// TIA Portal V19 export
FUNCTION "CEB_2" : Void   // FC15, LAD
{ S7_Optimized_Access := 'TRUE' }
// stored: SetENOAutomatically false
BEGIN

REGION Network 2: CEB_2 START
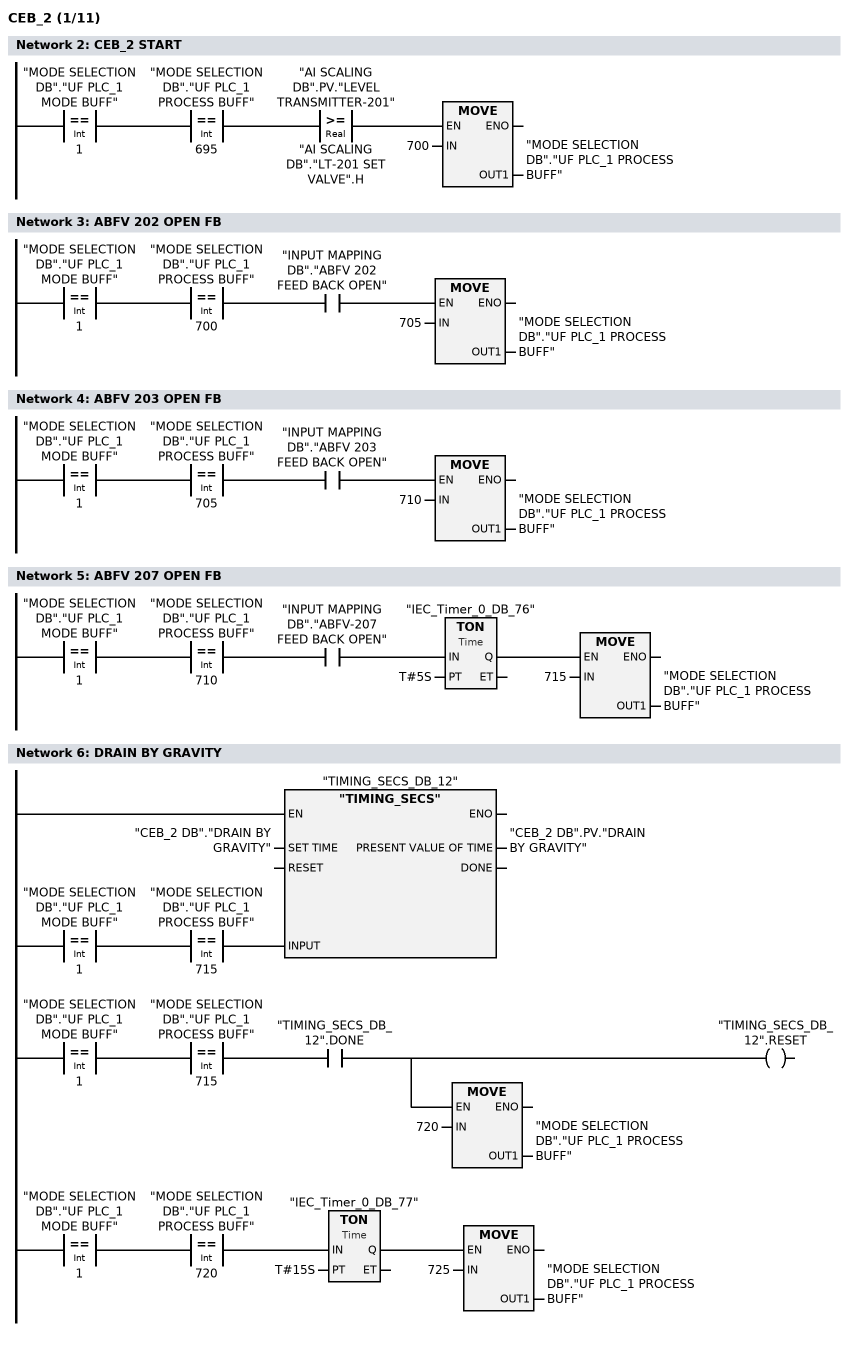
   RUNG wire#powerrail
      { S7_Templates := "SrcType := Int" } EQ_Contact(in1 := "MODE SELECTION DB"."UF PLC_1 MODE BUFF", in2 := 1)
      { S7_Templates := "SrcType := Int" } EQ_Contact(in1 := "MODE SELECTION DB"."UF PLC_1 PROCESS BUFF", in2 := 695)
      { S7_Templates := "SrcType := Real" } GE_Contact(in1 := "AI SCALING DB".PV."LEVEL TRANSMITTER-201", in2 := "AI SCALING DB"."LT-201 SET VALVE".H)
      Move(in := 700, out1 => "MODE SELECTION DB"."UF PLC_1 PROCESS BUFF")
   END_RUNG
   // the same network as SCL:
   IF ("MODE SELECTION DB"."UF PLC_1 MODE BUFF" = 1) AND ("MODE SELECTION DB"."UF PLC_1 PROCESS BUFF" = 695) AND ("AI SCALING DB".PV."LEVEL TRANSMITTER-201" >= "AI SCALING DB"."LT-201 SET VALVE".H) THEN
       "MODE SELECTION DB"."UF PLC_1 PROCESS BUFF" := 700;
   END_IF;
END_REGION

REGION Network 3: ABFV 202 OPEN FB
   RUNG wire#powerrail
      { S7_Templates := "SrcType := Int" } EQ_Contact(in1 := "MODE SELECTION DB"."UF PLC_1 MODE BUFF", in2 := 1)
      { S7_Templates := "SrcType := Int" } EQ_Contact(in1 := "MODE SELECTION DB"."UF PLC_1 PROCESS BUFF", in2 := 700)
      Contact( "INPUT MAPPING DB"."ABFV 202 FEED BACK OPEN" )
      Move(in := 705, out1 => "MODE SELECTION DB"."UF PLC_1 PROCESS BUFF")
   END_RUNG
   // the same network as SCL:
   IF ("MODE SELECTION DB"."UF PLC_1 MODE BUFF" = 1) AND ("MODE SELECTION DB"."UF PLC_1 PROCESS BUFF" = 700) AND "INPUT MAPPING DB"."ABFV 202 FEED BACK OPEN" THEN
       "MODE SELECTION DB"."UF PLC_1 PROCESS BUFF" := 705;
   END_IF;
END_REGION

REGION Network 4: ABFV 203 OPEN FB
   RUNG wire#powerrail
      { S7_Templates := "SrcType := Int" } EQ_Contact(in1 := "MODE SELECTION DB"."UF PLC_1 MODE BUFF", in2 := 1)
      { S7_Templates := "SrcType := Int" } EQ_Contact(in1 := "MODE SELECTION DB"."UF PLC_1 PROCESS BUFF", in2 := 705)
      Contact( "INPUT MAPPING DB"."ABFV 203 FEED BACK OPEN" )
      Move(in := 710, out1 => "MODE SELECTION DB"."UF PLC_1 PROCESS BUFF")
   END_RUNG
   // the same network as SCL:
   IF ("MODE SELECTION DB"."UF PLC_1 MODE BUFF" = 1) AND ("MODE SELECTION DB"."UF PLC_1 PROCESS BUFF" = 705) AND "INPUT MAPPING DB"."ABFV 203 FEED BACK OPEN" THEN
       "MODE SELECTION DB"."UF PLC_1 PROCESS BUFF" := 710;
   END_IF;
END_REGION

REGION Network 5: ABFV 207 OPEN FB
   RUNG wire#powerrail
      { S7_Templates := "SrcType := Int" } EQ_Contact(in1 := "MODE SELECTION DB"."UF PLC_1 MODE BUFF", in2 := 1)
      { S7_Templates := "SrcType := Int" } EQ_Contact(in1 := "MODE SELECTION DB"."UF PLC_1 PROCESS BUFF", in2 := 710)
      Contact( "INPUT MAPPING DB"."ABFV-207 FEED BACK OPEN" )
      { S7_Templates := "time_type := Time" } "IEC_Timer_0_DB_76".TON(pt := T#5S, et =>)
      Move(in := 715, out1 => "MODE SELECTION DB"."UF PLC_1 PROCESS BUFF")
   END_RUNG
   // the same network as SCL:
   "IEC_Timer_0_DB_76".TON(IN := ("MODE SELECTION DB"."UF PLC_1 MODE BUFF" = 1) AND ("MODE SELECTION DB"."UF PLC_1 PROCESS BUFF" = 710) AND "INPUT MAPPING DB"."ABFV-207 FEED BACK OPEN",
                           PT := T#5S);
   IF "IEC_Timer_0_DB_76".Q THEN "MODE SELECTION DB"."UF PLC_1 PROCESS BUFF" := 715; END_IF;
END_REGION

REGION Network 6: DRAIN BY GRAVITY
   RUNG wire#powerrail
      "TIMING_SECS_DB_12"(INPUT := wire#w1, "SET TIME" := "CEB_2 DB"."DRAIN BY GRAVITY", RESET :=, "PRESENT VALUE OF TIME" => "CEB_2 DB".PV."DRAIN BY GRAVITY", DONE =>)
   END_RUNG
   RUNG wire#powerrail
      { S7_Templates := "SrcType := Int" } EQ_Contact(in1 := "MODE SELECTION DB"."UF PLC_1 MODE BUFF", in2 := 1)
      { S7_Templates := "SrcType := Int" } EQ_Contact(in1 := "MODE SELECTION DB"."UF PLC_1 PROCESS BUFF", in2 := 715)
   END_RUNG wire#w1
   RUNG wire#powerrail
      { S7_Templates := "SrcType := Int" } EQ_Contact(in1 := "MODE SELECTION DB"."UF PLC_1 MODE BUFF", in2 := 1)
      { S7_Templates := "SrcType := Int" } EQ_Contact(in1 := "MODE SELECTION DB"."UF PLC_1 PROCESS BUFF", in2 := 715)
      Contact( "TIMING_SECS_DB_12".DONE )
      wire#w2
      Coil( "TIMING_SECS_DB_12".RESET )
   END_RUNG
   RUNG wire#w2
      Move(in := 720, out1 => "MODE SELECTION DB"."UF PLC_1 PROCESS BUFF")
   END_RUNG
   RUNG wire#powerrail
      { S7_Templates := "SrcType := Int" } EQ_Contact(in1 := "MODE SELECTION DB"."UF PLC_1 MODE BUFF", in2 := 1)
      { S7_Templates := "SrcType := Int" } EQ_Contact(in1 := "MODE SELECTION DB"."UF PLC_1 PROCESS BUFF", in2 := 720)
      { S7_Templates := "time_type := Time" } "IEC_Timer_0_DB_77".TON(pt := T#15S, et =>)
      Move(in := 725, out1 => "MODE SELECTION DB"."UF PLC_1 PROCESS BUFF")
   END_RUNG
   // the same network as SCL:
   "TIMING_SECS_DB_12"("SET TIME" := "CEB_2 DB"."DRAIN BY GRAVITY",   // "TIMING_SECS"
                       INPUT := ("MODE SELECTION DB"."UF PLC_1 MODE BUFF" = 1) AND ("MODE SELECTION DB"."UF PLC_1 PROCESS BUFF" = 715),
                       "PRESENT VALUE OF TIME" => "CEB_2 DB".PV."DRAIN BY GRAVITY");
   "TIMING_SECS_DB_12".RESET := ("MODE SELECTION DB"."UF PLC_1 MODE BUFF" = 1) AND ("MODE SELECTION DB"."UF PLC_1 PROCESS BUFF" = 715) AND "TIMING_SECS_DB_12".DONE;
   IF "TIMING_SECS_DB_12".RESET THEN "MODE SELECTION DB"."UF PLC_1 PROCESS BUFF" := 720; END_IF;
   "IEC_Timer_0_DB_77".TON(IN := ("MODE SELECTION DB"."UF PLC_1 MODE BUFF" = 1) AND ("MODE SELECTION DB"."UF PLC_1 PROCESS BUFF" = 720),
                           PT := T#15S);
   IF "IEC_Timer_0_DB_77".Q THEN "MODE SELECTION DB"."UF PLC_1 PROCESS BUFF" := 725; END_IF;
END_REGION

REGION Network 7: ABFV 207 CLOSE FB
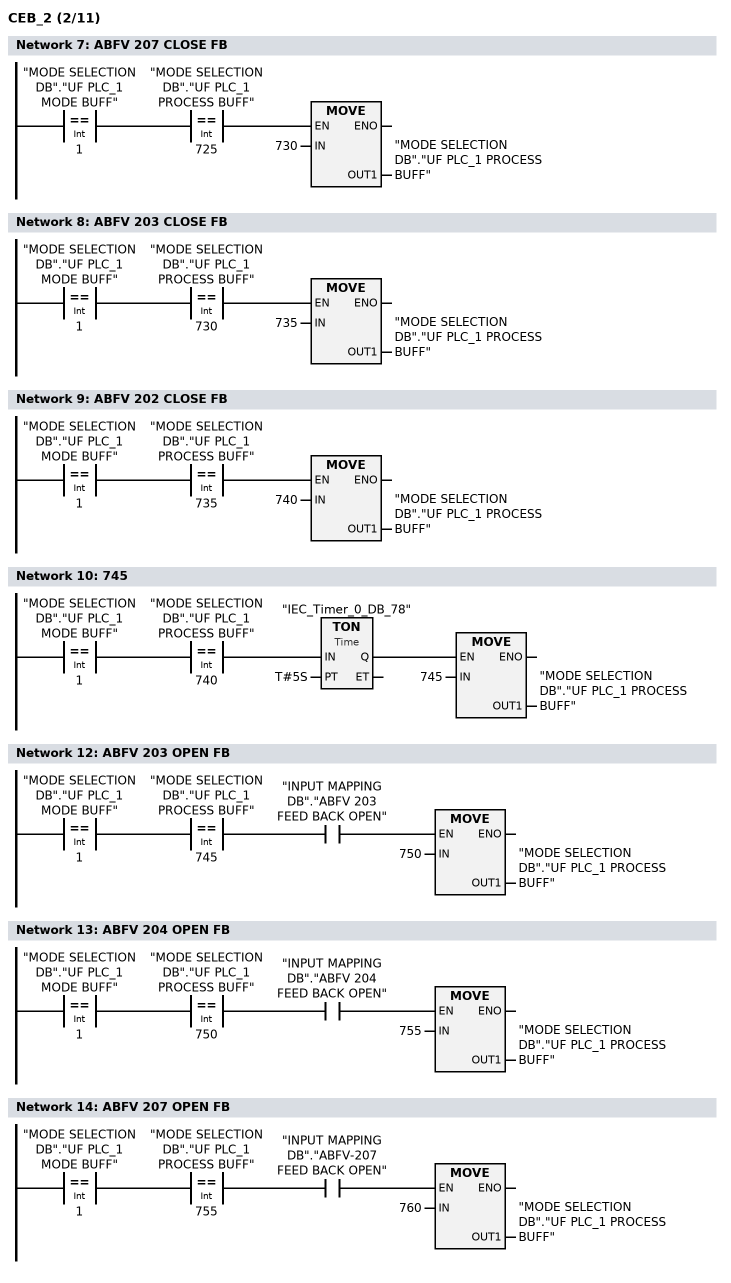
   RUNG wire#powerrail
      { S7_Templates := "SrcType := Int" } EQ_Contact(in1 := "MODE SELECTION DB"."UF PLC_1 MODE BUFF", in2 := 1)
      { S7_Templates := "SrcType := Int" } EQ_Contact(in1 := "MODE SELECTION DB"."UF PLC_1 PROCESS BUFF", in2 := 725)
      Move(in := 730, out1 => "MODE SELECTION DB"."UF PLC_1 PROCESS BUFF")
   END_RUNG
   // the same network as SCL:
   IF ("MODE SELECTION DB"."UF PLC_1 MODE BUFF" = 1) AND ("MODE SELECTION DB"."UF PLC_1 PROCESS BUFF" = 725) THEN
       "MODE SELECTION DB"."UF PLC_1 PROCESS BUFF" := 730;
   END_IF;
END_REGION

REGION Network 8: ABFV 203 CLOSE FB
   RUNG wire#powerrail
      { S7_Templates := "SrcType := Int" } EQ_Contact(in1 := "MODE SELECTION DB"."UF PLC_1 MODE BUFF", in2 := 1)
      { S7_Templates := "SrcType := Int" } EQ_Contact(in1 := "MODE SELECTION DB"."UF PLC_1 PROCESS BUFF", in2 := 730)
      Move(in := 735, out1 => "MODE SELECTION DB"."UF PLC_1 PROCESS BUFF")
   END_RUNG
   // the same network as SCL:
   IF ("MODE SELECTION DB"."UF PLC_1 MODE BUFF" = 1) AND ("MODE SELECTION DB"."UF PLC_1 PROCESS BUFF" = 730) THEN
       "MODE SELECTION DB"."UF PLC_1 PROCESS BUFF" := 735;
   END_IF;
END_REGION

REGION Network 9: ABFV 202 CLOSE FB
   RUNG wire#powerrail
      { S7_Templates := "SrcType := Int" } EQ_Contact(in1 := "MODE SELECTION DB"."UF PLC_1 MODE BUFF", in2 := 1)
      { S7_Templates := "SrcType := Int" } EQ_Contact(in1 := "MODE SELECTION DB"."UF PLC_1 PROCESS BUFF", in2 := 735)
      Move(in := 740, out1 => "MODE SELECTION DB"."UF PLC_1 PROCESS BUFF")
   END_RUNG
   // the same network as SCL:
   IF ("MODE SELECTION DB"."UF PLC_1 MODE BUFF" = 1) AND ("MODE SELECTION DB"."UF PLC_1 PROCESS BUFF" = 735) THEN
       "MODE SELECTION DB"."UF PLC_1 PROCESS BUFF" := 740;
   END_IF;
END_REGION

REGION Network 10: 745
   RUNG wire#powerrail
      { S7_Templates := "SrcType := Int" } EQ_Contact(in1 := "MODE SELECTION DB"."UF PLC_1 MODE BUFF", in2 := 1)
      { S7_Templates := "SrcType := Int" } EQ_Contact(in1 := "MODE SELECTION DB"."UF PLC_1 PROCESS BUFF", in2 := 740)
      { S7_Templates := "time_type := Time" } "IEC_Timer_0_DB_78".TON(pt := T#5S, et =>)
      Move(in := 745, out1 => "MODE SELECTION DB"."UF PLC_1 PROCESS BUFF")
   END_RUNG
   // the same network as SCL:
   "IEC_Timer_0_DB_78".TON(IN := ("MODE SELECTION DB"."UF PLC_1 MODE BUFF" = 1) AND ("MODE SELECTION DB"."UF PLC_1 PROCESS BUFF" = 740),
                           PT := T#5S);
   IF "IEC_Timer_0_DB_78".Q THEN "MODE SELECTION DB"."UF PLC_1 PROCESS BUFF" := 745; END_IF;
END_REGION

REGION Network 12: ABFV 203 OPEN FB
   RUNG wire#powerrail
      { S7_Templates := "SrcType := Int" } EQ_Contact(in1 := "MODE SELECTION DB"."UF PLC_1 MODE BUFF", in2 := 1)
      { S7_Templates := "SrcType := Int" } EQ_Contact(in1 := "MODE SELECTION DB"."UF PLC_1 PROCESS BUFF", in2 := 745)
      Contact( "INPUT MAPPING DB"."ABFV 203 FEED BACK OPEN" )
      Move(in := 750, out1 => "MODE SELECTION DB"."UF PLC_1 PROCESS BUFF")
   END_RUNG
   // the same network as SCL:
   IF ("MODE SELECTION DB"."UF PLC_1 MODE BUFF" = 1) AND ("MODE SELECTION DB"."UF PLC_1 PROCESS BUFF" = 745) AND "INPUT MAPPING DB"."ABFV 203 FEED BACK OPEN" THEN
       "MODE SELECTION DB"."UF PLC_1 PROCESS BUFF" := 750;
   END_IF;
END_REGION

REGION Network 13: ABFV 204 OPEN FB
   RUNG wire#powerrail
      { S7_Templates := "SrcType := Int" } EQ_Contact(in1 := "MODE SELECTION DB"."UF PLC_1 MODE BUFF", in2 := 1)
      { S7_Templates := "SrcType := Int" } EQ_Contact(in1 := "MODE SELECTION DB"."UF PLC_1 PROCESS BUFF", in2 := 750)
      Contact( "INPUT MAPPING DB"."ABFV 204 FEED BACK OPEN" )
      Move(in := 755, out1 => "MODE SELECTION DB"."UF PLC_1 PROCESS BUFF")
   END_RUNG
   // the same network as SCL:
   IF ("MODE SELECTION DB"."UF PLC_1 MODE BUFF" = 1) AND ("MODE SELECTION DB"."UF PLC_1 PROCESS BUFF" = 750) AND "INPUT MAPPING DB"."ABFV 204 FEED BACK OPEN" THEN
       "MODE SELECTION DB"."UF PLC_1 PROCESS BUFF" := 755;
   END_IF;
END_REGION

REGION Network 14: ABFV 207 OPEN FB
   RUNG wire#powerrail
      { S7_Templates := "SrcType := Int" } EQ_Contact(in1 := "MODE SELECTION DB"."UF PLC_1 MODE BUFF", in2 := 1)
      { S7_Templates := "SrcType := Int" } EQ_Contact(in1 := "MODE SELECTION DB"."UF PLC_1 PROCESS BUFF", in2 := 755)
      Contact( "INPUT MAPPING DB"."ABFV-207 FEED BACK OPEN" )
      Move(in := 760, out1 => "MODE SELECTION DB"."UF PLC_1 PROCESS BUFF")
   END_RUNG
   // the same network as SCL:
   IF ("MODE SELECTION DB"."UF PLC_1 MODE BUFF" = 1) AND ("MODE SELECTION DB"."UF PLC_1 PROCESS BUFF" = 755) AND "INPUT MAPPING DB"."ABFV-207 FEED BACK OPEN" THEN
       "MODE SELECTION DB"."UF PLC_1 PROCESS BUFF" := 760;
   END_IF;
END_REGION

REGION Network 15: ABFV 208 OPEN FB
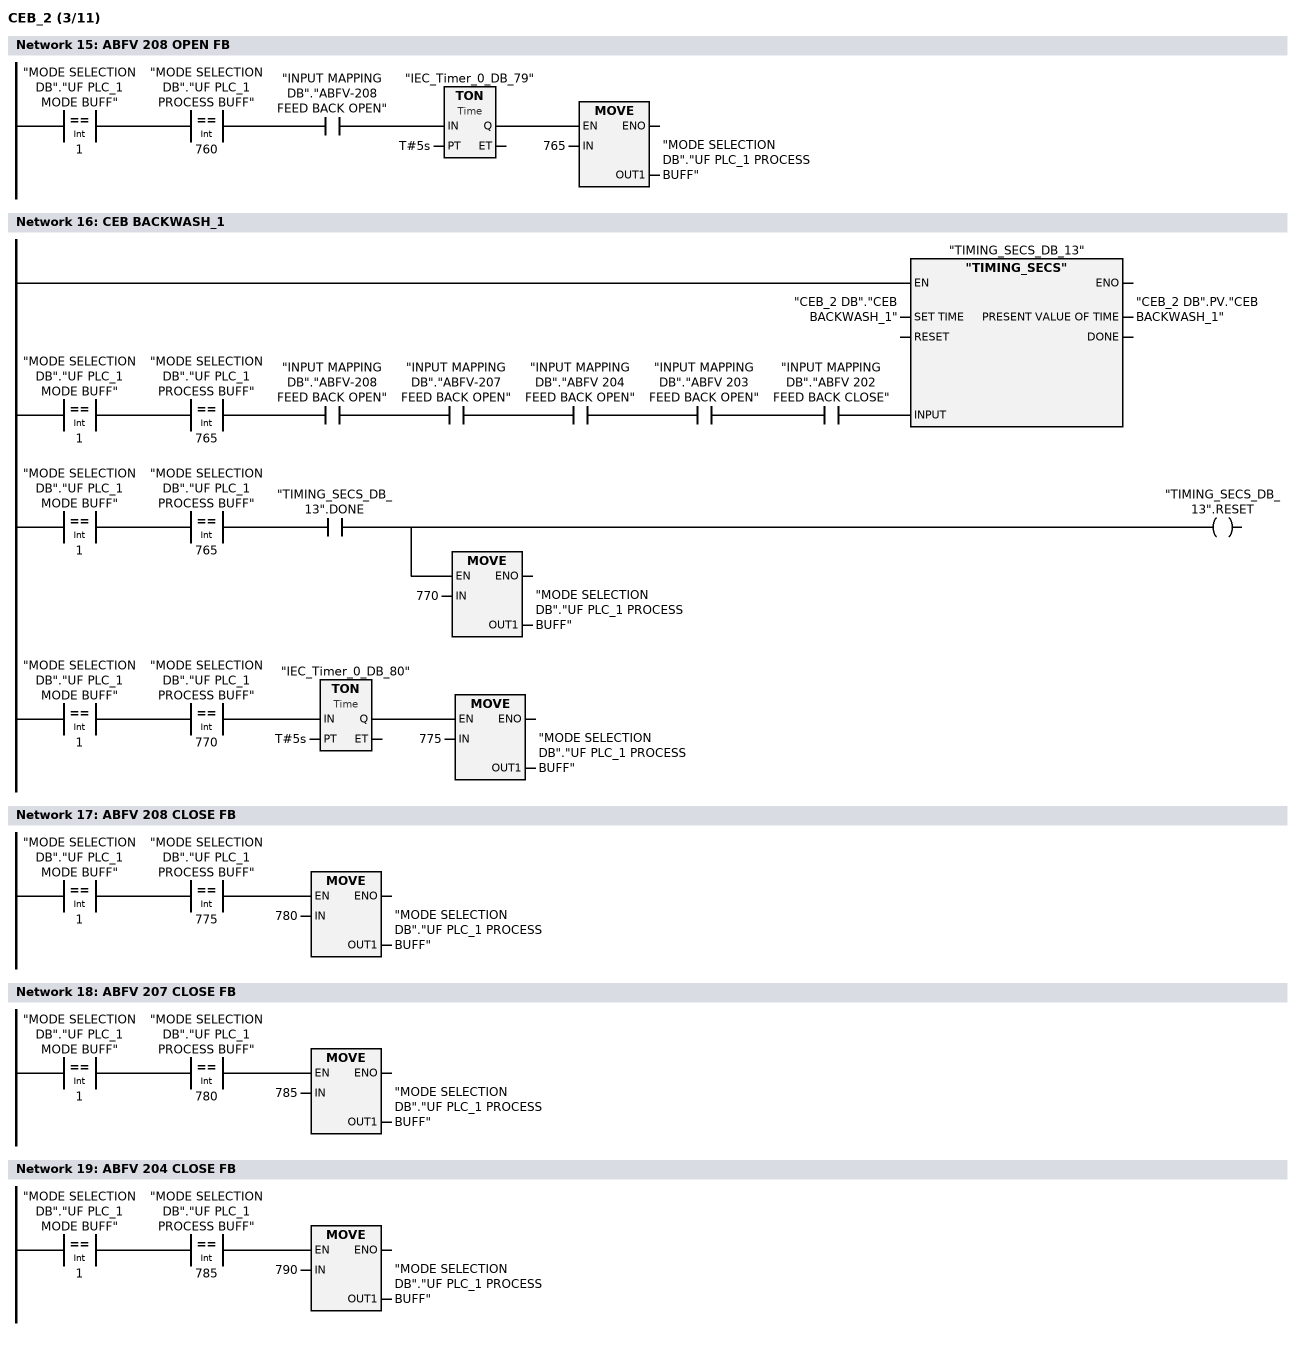
   RUNG wire#powerrail
      { S7_Templates := "SrcType := Int" } EQ_Contact(in1 := "MODE SELECTION DB"."UF PLC_1 MODE BUFF", in2 := 1)
      { S7_Templates := "SrcType := Int" } EQ_Contact(in1 := "MODE SELECTION DB"."UF PLC_1 PROCESS BUFF", in2 := 760)
      Contact( "INPUT MAPPING DB"."ABFV-208 FEED BACK OPEN" )
      { S7_Templates := "time_type := Time" } "IEC_Timer_0_DB_79".TON(pt := T#5s, et =>)
      Move(in := 765, out1 => "MODE SELECTION DB"."UF PLC_1 PROCESS BUFF")
   END_RUNG
   // the same network as SCL:
   "IEC_Timer_0_DB_79".TON(IN := ("MODE SELECTION DB"."UF PLC_1 MODE BUFF" = 1) AND ("MODE SELECTION DB"."UF PLC_1 PROCESS BUFF" = 760) AND "INPUT MAPPING DB"."ABFV-208 FEED BACK OPEN",
                           PT := T#5s);
   IF "IEC_Timer_0_DB_79".Q THEN "MODE SELECTION DB"."UF PLC_1 PROCESS BUFF" := 765; END_IF;
END_REGION

REGION Network 16: CEB BACKWASH_1
   RUNG wire#powerrail
      "TIMING_SECS_DB_13"(INPUT := wire#w1, "SET TIME" := "CEB_2 DB"."CEB BACKWASH_1", RESET :=, "PRESENT VALUE OF TIME" => "CEB_2 DB".PV."CEB BACKWASH_1", DONE =>)
   END_RUNG
   RUNG wire#powerrail
      { S7_Templates := "SrcType := Int" } EQ_Contact(in1 := "MODE SELECTION DB"."UF PLC_1 MODE BUFF", in2 := 1)
      { S7_Templates := "SrcType := Int" } EQ_Contact(in1 := "MODE SELECTION DB"."UF PLC_1 PROCESS BUFF", in2 := 765)
      Contact( "INPUT MAPPING DB"."ABFV-208 FEED BACK OPEN" )
      Contact( "INPUT MAPPING DB"."ABFV-207 FEED BACK OPEN" )
      Contact( "INPUT MAPPING DB"."ABFV 204 FEED BACK OPEN" )
      Contact( "INPUT MAPPING DB"."ABFV 203 FEED BACK OPEN" )
      Contact( "INPUT MAPPING DB"."ABFV 202 FEED BACK CLOSE" )
   END_RUNG wire#w1
   RUNG wire#powerrail
      { S7_Templates := "SrcType := Int" } EQ_Contact(in1 := "MODE SELECTION DB"."UF PLC_1 MODE BUFF", in2 := 1)
      { S7_Templates := "SrcType := Int" } EQ_Contact(in1 := "MODE SELECTION DB"."UF PLC_1 PROCESS BUFF", in2 := 765)
      Contact( "TIMING_SECS_DB_13".DONE )
      wire#w2
      Coil( "TIMING_SECS_DB_13".RESET )
   END_RUNG
   RUNG wire#w2
      Move(in := 770, out1 => "MODE SELECTION DB"."UF PLC_1 PROCESS BUFF")
   END_RUNG
   RUNG wire#powerrail
      { S7_Templates := "SrcType := Int" } EQ_Contact(in1 := "MODE SELECTION DB"."UF PLC_1 MODE BUFF", in2 := 1)
      { S7_Templates := "SrcType := Int" } EQ_Contact(in1 := "MODE SELECTION DB"."UF PLC_1 PROCESS BUFF", in2 := 770)
      { S7_Templates := "time_type := Time" } "IEC_Timer_0_DB_80".TON(pt := T#5s, et =>)
      Move(in := 775, out1 => "MODE SELECTION DB"."UF PLC_1 PROCESS BUFF")
   END_RUNG
   // the same network as SCL:
   "TIMING_SECS_DB_13"("SET TIME" := "CEB_2 DB"."CEB BACKWASH_1",   // "TIMING_SECS"
                       INPUT := ("MODE SELECTION DB"."UF PLC_1 MODE BUFF" = 1) AND ("MODE SELECTION DB"."UF PLC_1 PROCESS BUFF" = 765) AND "INPUT MAPPING DB"."ABFV-208 FEED BACK OPEN" AND "INPUT MAPPING DB"."ABFV-207 FEED BACK OPEN" AND "INPUT MAPPING DB"."ABFV 204 FEED BACK OPEN" AND "INPUT MAPPING DB"."ABFV 203 FEED BACK OPEN" AND "INPUT MAPPING DB"."ABFV 202 FEED BACK CLOSE",
                       "PRESENT VALUE OF TIME" => "CEB_2 DB".PV."CEB BACKWASH_1");
   "TIMING_SECS_DB_13".RESET := ("MODE SELECTION DB"."UF PLC_1 MODE BUFF" = 1) AND ("MODE SELECTION DB"."UF PLC_1 PROCESS BUFF" = 765) AND "TIMING_SECS_DB_13".DONE;
   IF "TIMING_SECS_DB_13".RESET THEN "MODE SELECTION DB"."UF PLC_1 PROCESS BUFF" := 770; END_IF;
   "IEC_Timer_0_DB_80".TON(IN := ("MODE SELECTION DB"."UF PLC_1 MODE BUFF" = 1) AND ("MODE SELECTION DB"."UF PLC_1 PROCESS BUFF" = 770),
                           PT := T#5s);
   IF "IEC_Timer_0_DB_80".Q THEN "MODE SELECTION DB"."UF PLC_1 PROCESS BUFF" := 775; END_IF;
END_REGION

REGION Network 17: ABFV 208 CLOSE FB
   RUNG wire#powerrail
      { S7_Templates := "SrcType := Int" } EQ_Contact(in1 := "MODE SELECTION DB"."UF PLC_1 MODE BUFF", in2 := 1)
      { S7_Templates := "SrcType := Int" } EQ_Contact(in1 := "MODE SELECTION DB"."UF PLC_1 PROCESS BUFF", in2 := 775)
      Move(in := 780, out1 => "MODE SELECTION DB"."UF PLC_1 PROCESS BUFF")
   END_RUNG
   // the same network as SCL:
   IF ("MODE SELECTION DB"."UF PLC_1 MODE BUFF" = 1) AND ("MODE SELECTION DB"."UF PLC_1 PROCESS BUFF" = 775) THEN
       "MODE SELECTION DB"."UF PLC_1 PROCESS BUFF" := 780;
   END_IF;
END_REGION

REGION Network 18: ABFV 207 CLOSE FB
   RUNG wire#powerrail
      { S7_Templates := "SrcType := Int" } EQ_Contact(in1 := "MODE SELECTION DB"."UF PLC_1 MODE BUFF", in2 := 1)
      { S7_Templates := "SrcType := Int" } EQ_Contact(in1 := "MODE SELECTION DB"."UF PLC_1 PROCESS BUFF", in2 := 780)
      Move(in := 785, out1 => "MODE SELECTION DB"."UF PLC_1 PROCESS BUFF")
   END_RUNG
   // the same network as SCL:
   IF ("MODE SELECTION DB"."UF PLC_1 MODE BUFF" = 1) AND ("MODE SELECTION DB"."UF PLC_1 PROCESS BUFF" = 780) THEN
       "MODE SELECTION DB"."UF PLC_1 PROCESS BUFF" := 785;
   END_IF;
END_REGION

REGION Network 19: ABFV 204 CLOSE FB
   RUNG wire#powerrail
      { S7_Templates := "SrcType := Int" } EQ_Contact(in1 := "MODE SELECTION DB"."UF PLC_1 MODE BUFF", in2 := 1)
      { S7_Templates := "SrcType := Int" } EQ_Contact(in1 := "MODE SELECTION DB"."UF PLC_1 PROCESS BUFF", in2 := 785)
      Move(in := 790, out1 => "MODE SELECTION DB"."UF PLC_1 PROCESS BUFF")
   END_RUNG
   // the same network as SCL:
   IF ("MODE SELECTION DB"."UF PLC_1 MODE BUFF" = 1) AND ("MODE SELECTION DB"."UF PLC_1 PROCESS BUFF" = 785) THEN
       "MODE SELECTION DB"."UF PLC_1 PROCESS BUFF" := 790;
   END_IF;
END_REGION

REGION Network 20: ABFV 203 CLOSE FB
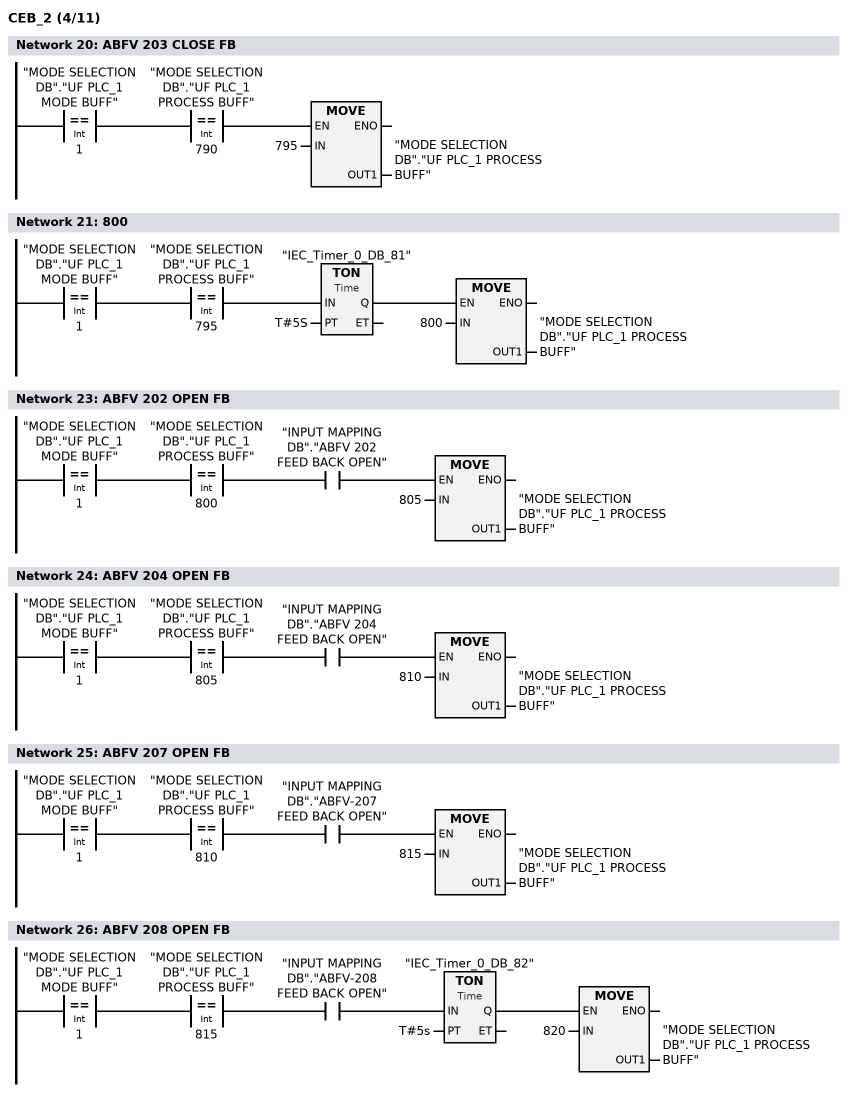
   RUNG wire#powerrail
      { S7_Templates := "SrcType := Int" } EQ_Contact(in1 := "MODE SELECTION DB"."UF PLC_1 MODE BUFF", in2 := 1)
      { S7_Templates := "SrcType := Int" } EQ_Contact(in1 := "MODE SELECTION DB"."UF PLC_1 PROCESS BUFF", in2 := 790)
      Move(in := 795, out1 => "MODE SELECTION DB"."UF PLC_1 PROCESS BUFF")
   END_RUNG
   // the same network as SCL:
   IF ("MODE SELECTION DB"."UF PLC_1 MODE BUFF" = 1) AND ("MODE SELECTION DB"."UF PLC_1 PROCESS BUFF" = 790) THEN
       "MODE SELECTION DB"."UF PLC_1 PROCESS BUFF" := 795;
   END_IF;
END_REGION

REGION Network 21: 800
   RUNG wire#powerrail
      { S7_Templates := "SrcType := Int" } EQ_Contact(in1 := "MODE SELECTION DB"."UF PLC_1 MODE BUFF", in2 := 1)
      { S7_Templates := "SrcType := Int" } EQ_Contact(in1 := "MODE SELECTION DB"."UF PLC_1 PROCESS BUFF", in2 := 795)
      { S7_Templates := "time_type := Time" } "IEC_Timer_0_DB_81".TON(pt := T#5S, et =>)
      Move(in := 800, out1 => "MODE SELECTION DB"."UF PLC_1 PROCESS BUFF")
   END_RUNG
   // the same network as SCL:
   "IEC_Timer_0_DB_81".TON(IN := ("MODE SELECTION DB"."UF PLC_1 MODE BUFF" = 1) AND ("MODE SELECTION DB"."UF PLC_1 PROCESS BUFF" = 795),
                           PT := T#5S);
   IF "IEC_Timer_0_DB_81".Q THEN "MODE SELECTION DB"."UF PLC_1 PROCESS BUFF" := 800; END_IF;
END_REGION

REGION Network 23: ABFV 202 OPEN FB
   RUNG wire#powerrail
      { S7_Templates := "SrcType := Int" } EQ_Contact(in1 := "MODE SELECTION DB"."UF PLC_1 MODE BUFF", in2 := 1)
      { S7_Templates := "SrcType := Int" } EQ_Contact(in1 := "MODE SELECTION DB"."UF PLC_1 PROCESS BUFF", in2 := 800)
      Contact( "INPUT MAPPING DB"."ABFV 202 FEED BACK OPEN" )
      Move(in := 805, out1 => "MODE SELECTION DB"."UF PLC_1 PROCESS BUFF")
   END_RUNG
   // the same network as SCL:
   IF ("MODE SELECTION DB"."UF PLC_1 MODE BUFF" = 1) AND ("MODE SELECTION DB"."UF PLC_1 PROCESS BUFF" = 800) AND "INPUT MAPPING DB"."ABFV 202 FEED BACK OPEN" THEN
       "MODE SELECTION DB"."UF PLC_1 PROCESS BUFF" := 805;
   END_IF;
END_REGION

REGION Network 24: ABFV 204 OPEN FB
   RUNG wire#powerrail
      { S7_Templates := "SrcType := Int" } EQ_Contact(in1 := "MODE SELECTION DB"."UF PLC_1 MODE BUFF", in2 := 1)
      { S7_Templates := "SrcType := Int" } EQ_Contact(in1 := "MODE SELECTION DB"."UF PLC_1 PROCESS BUFF", in2 := 805)
      Contact( "INPUT MAPPING DB"."ABFV 204 FEED BACK OPEN" )
      Move(in := 810, out1 => "MODE SELECTION DB"."UF PLC_1 PROCESS BUFF")
   END_RUNG
   // the same network as SCL:
   IF ("MODE SELECTION DB"."UF PLC_1 MODE BUFF" = 1) AND ("MODE SELECTION DB"."UF PLC_1 PROCESS BUFF" = 805) AND "INPUT MAPPING DB"."ABFV 204 FEED BACK OPEN" THEN
       "MODE SELECTION DB"."UF PLC_1 PROCESS BUFF" := 810;
   END_IF;
END_REGION

REGION Network 25: ABFV 207 OPEN FB
   RUNG wire#powerrail
      { S7_Templates := "SrcType := Int" } EQ_Contact(in1 := "MODE SELECTION DB"."UF PLC_1 MODE BUFF", in2 := 1)
      { S7_Templates := "SrcType := Int" } EQ_Contact(in1 := "MODE SELECTION DB"."UF PLC_1 PROCESS BUFF", in2 := 810)
      Contact( "INPUT MAPPING DB"."ABFV-207 FEED BACK OPEN" )
      Move(in := 815, out1 => "MODE SELECTION DB"."UF PLC_1 PROCESS BUFF")
   END_RUNG
   // the same network as SCL:
   IF ("MODE SELECTION DB"."UF PLC_1 MODE BUFF" = 1) AND ("MODE SELECTION DB"."UF PLC_1 PROCESS BUFF" = 810) AND "INPUT MAPPING DB"."ABFV-207 FEED BACK OPEN" THEN
       "MODE SELECTION DB"."UF PLC_1 PROCESS BUFF" := 815;
   END_IF;
END_REGION

REGION Network 26: ABFV 208 OPEN FB
   RUNG wire#powerrail
      { S7_Templates := "SrcType := Int" } EQ_Contact(in1 := "MODE SELECTION DB"."UF PLC_1 MODE BUFF", in2 := 1)
      { S7_Templates := "SrcType := Int" } EQ_Contact(in1 := "MODE SELECTION DB"."UF PLC_1 PROCESS BUFF", in2 := 815)
      Contact( "INPUT MAPPING DB"."ABFV-208 FEED BACK OPEN" )
      { S7_Templates := "time_type := Time" } "IEC_Timer_0_DB_82".TON(pt := T#5s, et =>)
      Move(in := 820, out1 => "MODE SELECTION DB"."UF PLC_1 PROCESS BUFF")
   END_RUNG
   // the same network as SCL:
   "IEC_Timer_0_DB_82".TON(IN := ("MODE SELECTION DB"."UF PLC_1 MODE BUFF" = 1) AND ("MODE SELECTION DB"."UF PLC_1 PROCESS BUFF" = 815) AND "INPUT MAPPING DB"."ABFV-208 FEED BACK OPEN",
                           PT := T#5s);
   IF "IEC_Timer_0_DB_82".Q THEN "MODE SELECTION DB"."UF PLC_1 PROCESS BUFF" := 820; END_IF;
END_REGION

REGION Network 27: CEB BACKWASH_2
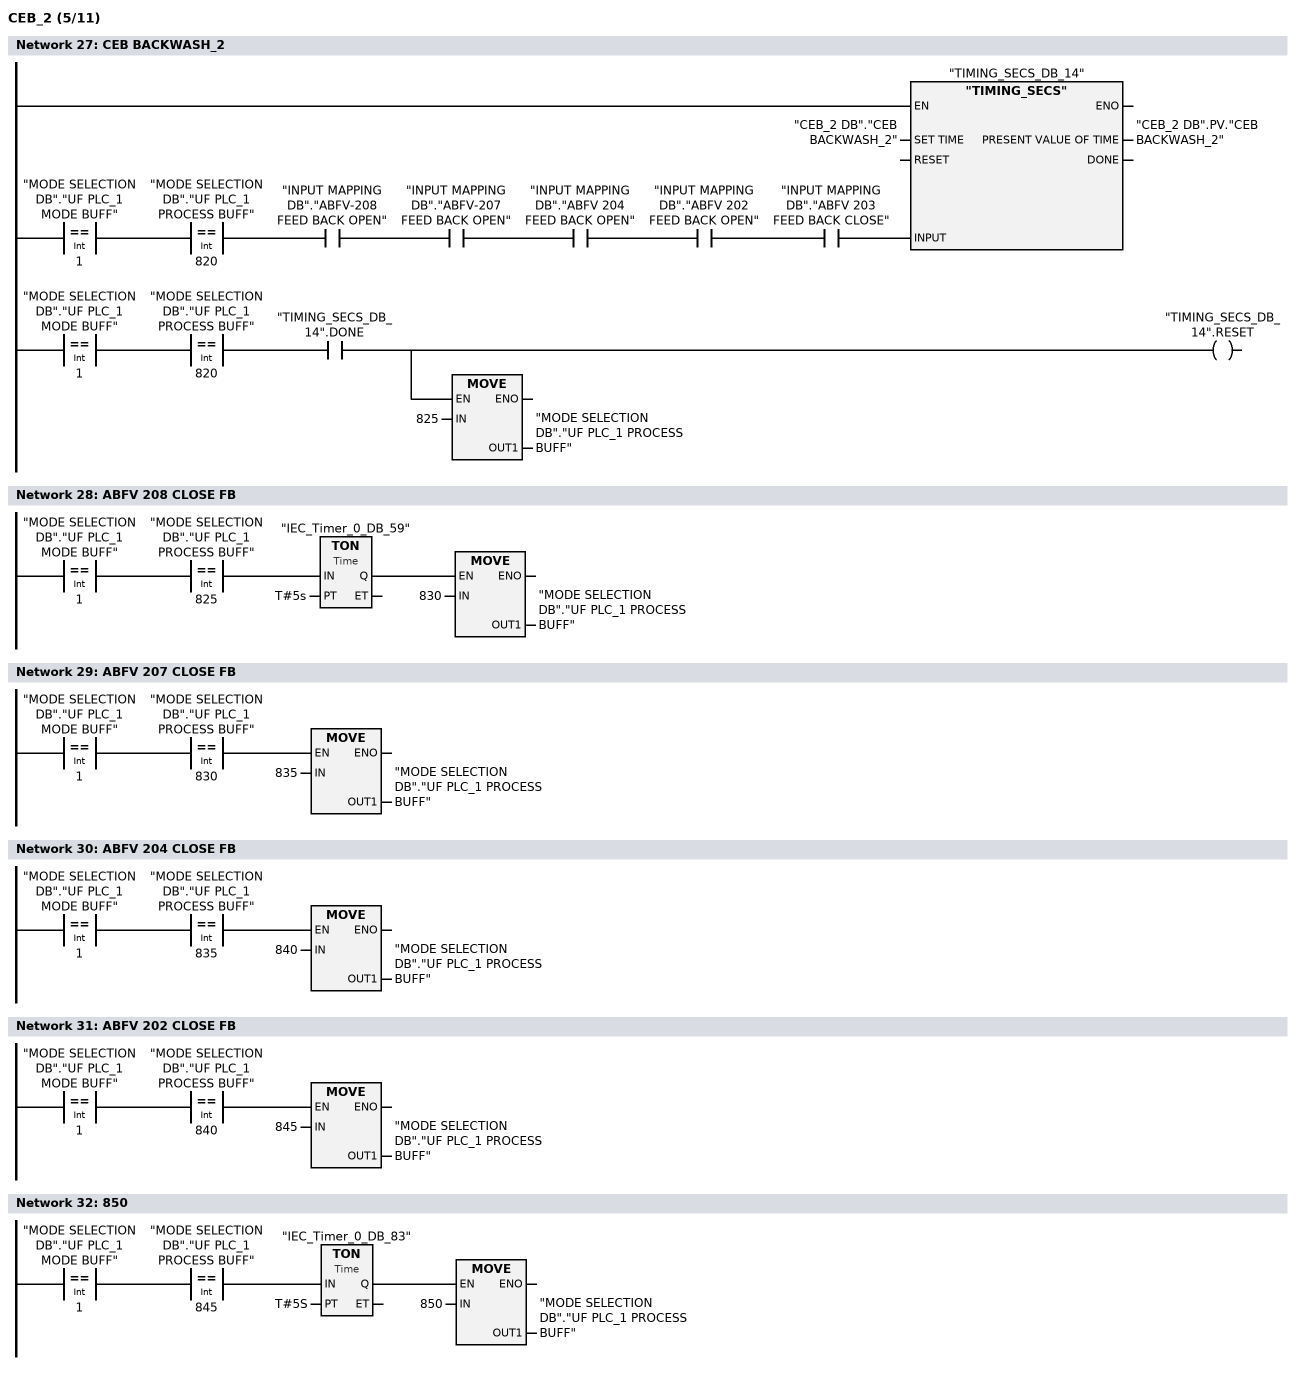
   RUNG wire#powerrail
      "TIMING_SECS_DB_14"(INPUT := wire#w1, "SET TIME" := "CEB_2 DB"."CEB BACKWASH_2", RESET :=, "PRESENT VALUE OF TIME" => "CEB_2 DB".PV."CEB BACKWASH_2", DONE =>)
   END_RUNG
   RUNG wire#powerrail
      { S7_Templates := "SrcType := Int" } EQ_Contact(in1 := "MODE SELECTION DB"."UF PLC_1 MODE BUFF", in2 := 1)
      { S7_Templates := "SrcType := Int" } EQ_Contact(in1 := "MODE SELECTION DB"."UF PLC_1 PROCESS BUFF", in2 := 820)
      Contact( "INPUT MAPPING DB"."ABFV-208 FEED BACK OPEN" )
      Contact( "INPUT MAPPING DB"."ABFV-207 FEED BACK OPEN" )
      Contact( "INPUT MAPPING DB"."ABFV 204 FEED BACK OPEN" )
      Contact( "INPUT MAPPING DB"."ABFV 202 FEED BACK OPEN" )
      Contact( "INPUT MAPPING DB"."ABFV 203 FEED BACK CLOSE" )
   END_RUNG wire#w1
   RUNG wire#powerrail
      { S7_Templates := "SrcType := Int" } EQ_Contact(in1 := "MODE SELECTION DB"."UF PLC_1 MODE BUFF", in2 := 1)
      { S7_Templates := "SrcType := Int" } EQ_Contact(in1 := "MODE SELECTION DB"."UF PLC_1 PROCESS BUFF", in2 := 820)
      Contact( "TIMING_SECS_DB_14".DONE )
      wire#w2
      Coil( "TIMING_SECS_DB_14".RESET )
   END_RUNG
   RUNG wire#w2
      Move(in := 825, out1 => "MODE SELECTION DB"."UF PLC_1 PROCESS BUFF")
   END_RUNG
   // the same network as SCL:
   "TIMING_SECS_DB_14"("SET TIME" := "CEB_2 DB"."CEB BACKWASH_2",   // "TIMING_SECS"
                       INPUT := ("MODE SELECTION DB"."UF PLC_1 MODE BUFF" = 1) AND ("MODE SELECTION DB"."UF PLC_1 PROCESS BUFF" = 820) AND "INPUT MAPPING DB"."ABFV-208 FEED BACK OPEN" AND "INPUT MAPPING DB"."ABFV-207 FEED BACK OPEN" AND "INPUT MAPPING DB"."ABFV 204 FEED BACK OPEN" AND "INPUT MAPPING DB"."ABFV 202 FEED BACK OPEN" AND "INPUT MAPPING DB"."ABFV 203 FEED BACK CLOSE",
                       "PRESENT VALUE OF TIME" => "CEB_2 DB".PV."CEB BACKWASH_2");
   "TIMING_SECS_DB_14".RESET := ("MODE SELECTION DB"."UF PLC_1 MODE BUFF" = 1) AND ("MODE SELECTION DB"."UF PLC_1 PROCESS BUFF" = 820) AND "TIMING_SECS_DB_14".DONE;
   IF "TIMING_SECS_DB_14".RESET THEN "MODE SELECTION DB"."UF PLC_1 PROCESS BUFF" := 825; END_IF;
END_REGION

REGION Network 28: ABFV 208 CLOSE FB
   RUNG wire#powerrail
      { S7_Templates := "SrcType := Int" } EQ_Contact(in1 := "MODE SELECTION DB"."UF PLC_1 MODE BUFF", in2 := 1)
      { S7_Templates := "SrcType := Int" } EQ_Contact(in1 := "MODE SELECTION DB"."UF PLC_1 PROCESS BUFF", in2 := 825)
      { S7_Templates := "time_type := Time" } "IEC_Timer_0_DB_59".TON(pt := T#5s, et =>)
      Move(in := 830, out1 => "MODE SELECTION DB"."UF PLC_1 PROCESS BUFF")
   END_RUNG
   // the same network as SCL:
   "IEC_Timer_0_DB_59".TON(IN := ("MODE SELECTION DB"."UF PLC_1 MODE BUFF" = 1) AND ("MODE SELECTION DB"."UF PLC_1 PROCESS BUFF" = 825),
                           PT := T#5s);
   IF "IEC_Timer_0_DB_59".Q THEN "MODE SELECTION DB"."UF PLC_1 PROCESS BUFF" := 830; END_IF;
END_REGION

REGION Network 29: ABFV 207 CLOSE FB
   RUNG wire#powerrail
      { S7_Templates := "SrcType := Int" } EQ_Contact(in1 := "MODE SELECTION DB"."UF PLC_1 MODE BUFF", in2 := 1)
      { S7_Templates := "SrcType := Int" } EQ_Contact(in1 := "MODE SELECTION DB"."UF PLC_1 PROCESS BUFF", in2 := 830)
      Move(in := 835, out1 => "MODE SELECTION DB"."UF PLC_1 PROCESS BUFF")
   END_RUNG
   // the same network as SCL:
   IF ("MODE SELECTION DB"."UF PLC_1 MODE BUFF" = 1) AND ("MODE SELECTION DB"."UF PLC_1 PROCESS BUFF" = 830) THEN
       "MODE SELECTION DB"."UF PLC_1 PROCESS BUFF" := 835;
   END_IF;
END_REGION

REGION Network 30: ABFV 204 CLOSE FB
   RUNG wire#powerrail
      { S7_Templates := "SrcType := Int" } EQ_Contact(in1 := "MODE SELECTION DB"."UF PLC_1 MODE BUFF", in2 := 1)
      { S7_Templates := "SrcType := Int" } EQ_Contact(in1 := "MODE SELECTION DB"."UF PLC_1 PROCESS BUFF", in2 := 835)
      Move(in := 840, out1 => "MODE SELECTION DB"."UF PLC_1 PROCESS BUFF")
   END_RUNG
   // the same network as SCL:
   IF ("MODE SELECTION DB"."UF PLC_1 MODE BUFF" = 1) AND ("MODE SELECTION DB"."UF PLC_1 PROCESS BUFF" = 835) THEN
       "MODE SELECTION DB"."UF PLC_1 PROCESS BUFF" := 840;
   END_IF;
END_REGION

REGION Network 31: ABFV 202 CLOSE FB
   RUNG wire#powerrail
      { S7_Templates := "SrcType := Int" } EQ_Contact(in1 := "MODE SELECTION DB"."UF PLC_1 MODE BUFF", in2 := 1)
      { S7_Templates := "SrcType := Int" } EQ_Contact(in1 := "MODE SELECTION DB"."UF PLC_1 PROCESS BUFF", in2 := 840)
      Move(in := 845, out1 => "MODE SELECTION DB"."UF PLC_1 PROCESS BUFF")
   END_RUNG
   // the same network as SCL:
   IF ("MODE SELECTION DB"."UF PLC_1 MODE BUFF" = 1) AND ("MODE SELECTION DB"."UF PLC_1 PROCESS BUFF" = 840) THEN
       "MODE SELECTION DB"."UF PLC_1 PROCESS BUFF" := 845;
   END_IF;
END_REGION

REGION Network 32: 850
   RUNG wire#powerrail
      { S7_Templates := "SrcType := Int" } EQ_Contact(in1 := "MODE SELECTION DB"."UF PLC_1 MODE BUFF", in2 := 1)
      { S7_Templates := "SrcType := Int" } EQ_Contact(in1 := "MODE SELECTION DB"."UF PLC_1 PROCESS BUFF", in2 := 845)
      { S7_Templates := "time_type := Time" } "IEC_Timer_0_DB_83".TON(pt := T#5S, et =>)
      Move(in := 850, out1 => "MODE SELECTION DB"."UF PLC_1 PROCESS BUFF")
   END_RUNG
   // the same network as SCL:
   "IEC_Timer_0_DB_83".TON(IN := ("MODE SELECTION DB"."UF PLC_1 MODE BUFF" = 1) AND ("MODE SELECTION DB"."UF PLC_1 PROCESS BUFF" = 845),
                           PT := T#5S);
   IF "IEC_Timer_0_DB_83".Q THEN "MODE SELECTION DB"."UF PLC_1 PROCESS BUFF" := 850; END_IF;
END_REGION

REGION Network 34: SOAK
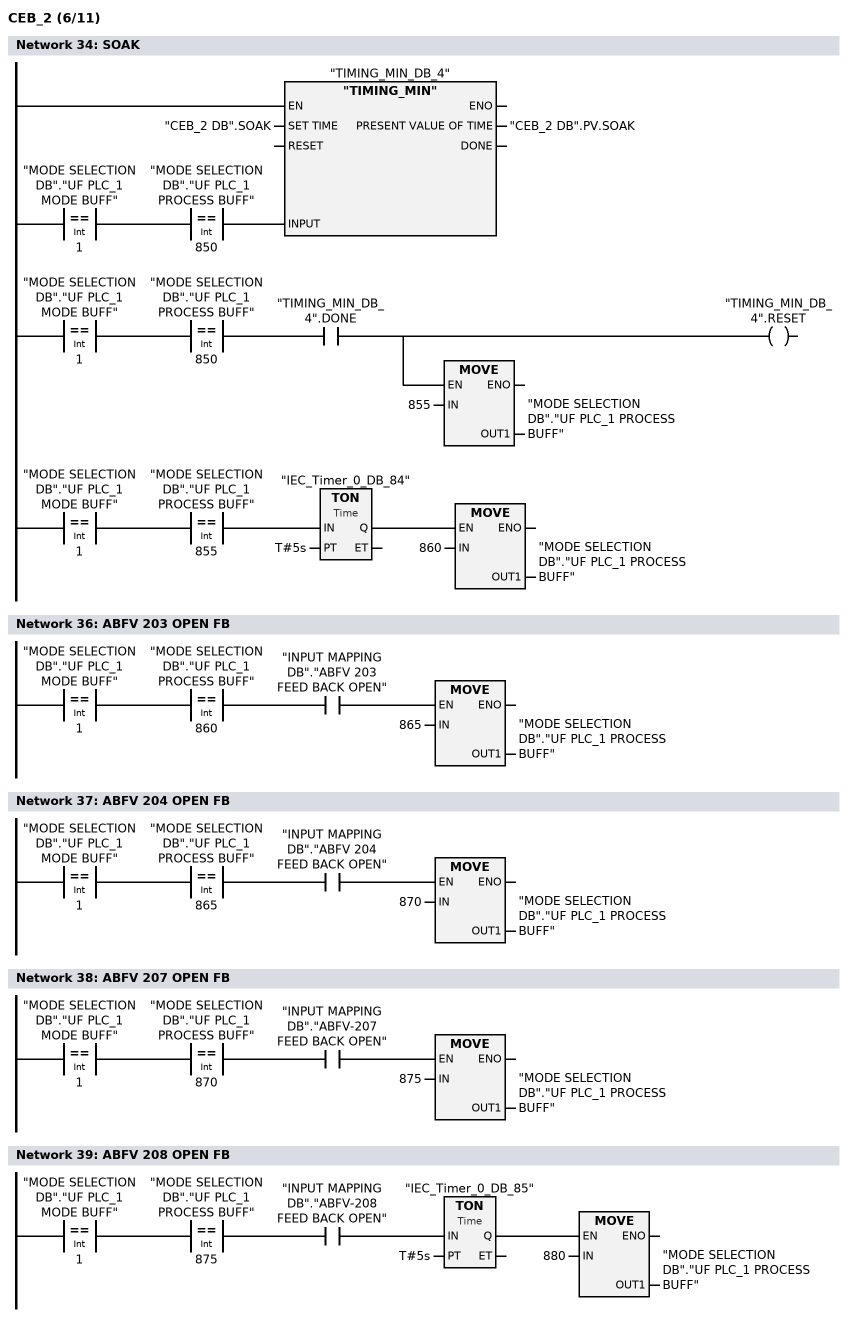
   RUNG wire#powerrail
      "TIMING_MIN_DB_4"(INPUT := wire#w1, "SET TIME" := "CEB_2 DB".SOAK, RESET :=, "PRESENT VALUE OF TIME" => "CEB_2 DB".PV.SOAK, DONE =>)
   END_RUNG
   RUNG wire#powerrail
      { S7_Templates := "SrcType := Int" } EQ_Contact(in1 := "MODE SELECTION DB"."UF PLC_1 MODE BUFF", in2 := 1)
      { S7_Templates := "SrcType := Int" } EQ_Contact(in1 := "MODE SELECTION DB"."UF PLC_1 PROCESS BUFF", in2 := 850)
   END_RUNG wire#w1
   RUNG wire#powerrail
      { S7_Templates := "SrcType := Int" } EQ_Contact(in1 := "MODE SELECTION DB"."UF PLC_1 MODE BUFF", in2 := 1)
      { S7_Templates := "SrcType := Int" } EQ_Contact(in1 := "MODE SELECTION DB"."UF PLC_1 PROCESS BUFF", in2 := 850)
      Contact( "TIMING_MIN_DB_4".DONE )
      wire#w2
      Coil( "TIMING_MIN_DB_4".RESET )
   END_RUNG
   RUNG wire#w2
      Move(in := 855, out1 => "MODE SELECTION DB"."UF PLC_1 PROCESS BUFF")
   END_RUNG
   RUNG wire#powerrail
      { S7_Templates := "SrcType := Int" } EQ_Contact(in1 := "MODE SELECTION DB"."UF PLC_1 MODE BUFF", in2 := 1)
      { S7_Templates := "SrcType := Int" } EQ_Contact(in1 := "MODE SELECTION DB"."UF PLC_1 PROCESS BUFF", in2 := 855)
      { S7_Templates := "time_type := Time" } "IEC_Timer_0_DB_84".TON(pt := T#5s, et =>)
      Move(in := 860, out1 => "MODE SELECTION DB"."UF PLC_1 PROCESS BUFF")
   END_RUNG
   // the same network as SCL:
   "TIMING_MIN_DB_4"("SET TIME" := "CEB_2 DB".SOAK,   // "TIMING_MIN"
                     INPUT := ("MODE SELECTION DB"."UF PLC_1 MODE BUFF" = 1) AND ("MODE SELECTION DB"."UF PLC_1 PROCESS BUFF" = 850),
                     "PRESENT VALUE OF TIME" => "CEB_2 DB".PV.SOAK);
   "TIMING_MIN_DB_4".RESET := ("MODE SELECTION DB"."UF PLC_1 MODE BUFF" = 1) AND ("MODE SELECTION DB"."UF PLC_1 PROCESS BUFF" = 850) AND "TIMING_MIN_DB_4".DONE;
   IF "TIMING_MIN_DB_4".RESET THEN "MODE SELECTION DB"."UF PLC_1 PROCESS BUFF" := 855; END_IF;
   "IEC_Timer_0_DB_84".TON(IN := ("MODE SELECTION DB"."UF PLC_1 MODE BUFF" = 1) AND ("MODE SELECTION DB"."UF PLC_1 PROCESS BUFF" = 855),
                           PT := T#5s);
   IF "IEC_Timer_0_DB_84".Q THEN "MODE SELECTION DB"."UF PLC_1 PROCESS BUFF" := 860; END_IF;
END_REGION

REGION Network 36: ABFV 203 OPEN FB
   RUNG wire#powerrail
      { S7_Templates := "SrcType := Int" } EQ_Contact(in1 := "MODE SELECTION DB"."UF PLC_1 MODE BUFF", in2 := 1)
      { S7_Templates := "SrcType := Int" } EQ_Contact(in1 := "MODE SELECTION DB"."UF PLC_1 PROCESS BUFF", in2 := 860)
      Contact( "INPUT MAPPING DB"."ABFV 203 FEED BACK OPEN" )
      Move(in := 865, out1 => "MODE SELECTION DB"."UF PLC_1 PROCESS BUFF")
   END_RUNG
   // the same network as SCL:
   IF ("MODE SELECTION DB"."UF PLC_1 MODE BUFF" = 1) AND ("MODE SELECTION DB"."UF PLC_1 PROCESS BUFF" = 860) AND "INPUT MAPPING DB"."ABFV 203 FEED BACK OPEN" THEN
       "MODE SELECTION DB"."UF PLC_1 PROCESS BUFF" := 865;
   END_IF;
END_REGION

REGION Network 37: ABFV 204 OPEN FB
   RUNG wire#powerrail
      { S7_Templates := "SrcType := Int" } EQ_Contact(in1 := "MODE SELECTION DB"."UF PLC_1 MODE BUFF", in2 := 1)
      { S7_Templates := "SrcType := Int" } EQ_Contact(in1 := "MODE SELECTION DB"."UF PLC_1 PROCESS BUFF", in2 := 865)
      Contact( "INPUT MAPPING DB"."ABFV 204 FEED BACK OPEN" )
      Move(in := 870, out1 => "MODE SELECTION DB"."UF PLC_1 PROCESS BUFF")
   END_RUNG
   // the same network as SCL:
   IF ("MODE SELECTION DB"."UF PLC_1 MODE BUFF" = 1) AND ("MODE SELECTION DB"."UF PLC_1 PROCESS BUFF" = 865) AND "INPUT MAPPING DB"."ABFV 204 FEED BACK OPEN" THEN
       "MODE SELECTION DB"."UF PLC_1 PROCESS BUFF" := 870;
   END_IF;
END_REGION

REGION Network 38: ABFV 207 OPEN FB
   RUNG wire#powerrail
      { S7_Templates := "SrcType := Int" } EQ_Contact(in1 := "MODE SELECTION DB"."UF PLC_1 MODE BUFF", in2 := 1)
      { S7_Templates := "SrcType := Int" } EQ_Contact(in1 := "MODE SELECTION DB"."UF PLC_1 PROCESS BUFF", in2 := 870)
      Contact( "INPUT MAPPING DB"."ABFV-207 FEED BACK OPEN" )
      Move(in := 875, out1 => "MODE SELECTION DB"."UF PLC_1 PROCESS BUFF")
   END_RUNG
   // the same network as SCL:
   IF ("MODE SELECTION DB"."UF PLC_1 MODE BUFF" = 1) AND ("MODE SELECTION DB"."UF PLC_1 PROCESS BUFF" = 870) AND "INPUT MAPPING DB"."ABFV-207 FEED BACK OPEN" THEN
       "MODE SELECTION DB"."UF PLC_1 PROCESS BUFF" := 875;
   END_IF;
END_REGION

REGION Network 39: ABFV 208 OPEN FB
   RUNG wire#powerrail
      { S7_Templates := "SrcType := Int" } EQ_Contact(in1 := "MODE SELECTION DB"."UF PLC_1 MODE BUFF", in2 := 1)
      { S7_Templates := "SrcType := Int" } EQ_Contact(in1 := "MODE SELECTION DB"."UF PLC_1 PROCESS BUFF", in2 := 875)
      Contact( "INPUT MAPPING DB"."ABFV-208 FEED BACK OPEN" )
      { S7_Templates := "time_type := Time" } "IEC_Timer_0_DB_85".TON(pt := T#5s, et =>)
      Move(in := 880, out1 => "MODE SELECTION DB"."UF PLC_1 PROCESS BUFF")
   END_RUNG
   // the same network as SCL:
   "IEC_Timer_0_DB_85".TON(IN := ("MODE SELECTION DB"."UF PLC_1 MODE BUFF" = 1) AND ("MODE SELECTION DB"."UF PLC_1 PROCESS BUFF" = 875) AND "INPUT MAPPING DB"."ABFV-208 FEED BACK OPEN",
                           PT := T#5s);
   IF "IEC_Timer_0_DB_85".Q THEN "MODE SELECTION DB"."UF PLC_1 PROCESS BUFF" := 880; END_IF;
END_REGION

REGION Network 40: BACKWASH_1
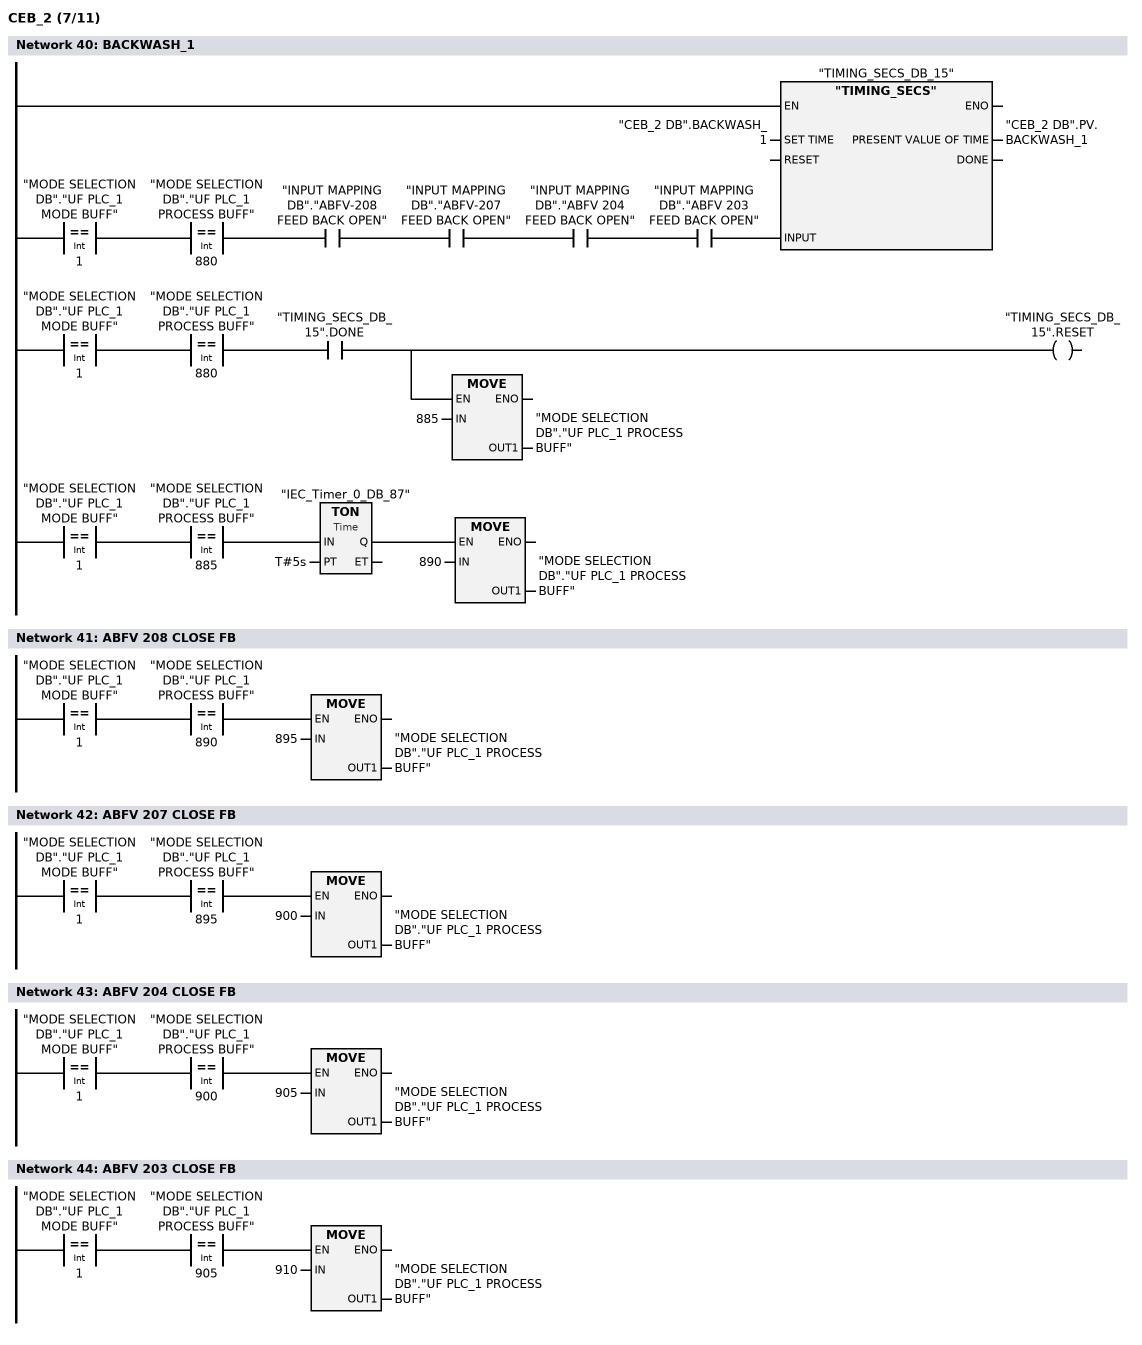
   RUNG wire#powerrail
      "TIMING_SECS_DB_15"(INPUT := wire#w1, "SET TIME" := "CEB_2 DB".BACKWASH_1, RESET :=, "PRESENT VALUE OF TIME" => "CEB_2 DB".PV.BACKWASH_1, DONE =>)
   END_RUNG
   RUNG wire#powerrail
      { S7_Templates := "SrcType := Int" } EQ_Contact(in1 := "MODE SELECTION DB"."UF PLC_1 MODE BUFF", in2 := 1)
      { S7_Templates := "SrcType := Int" } EQ_Contact(in1 := "MODE SELECTION DB"."UF PLC_1 PROCESS BUFF", in2 := 880)
      Contact( "INPUT MAPPING DB"."ABFV-208 FEED BACK OPEN" )
      Contact( "INPUT MAPPING DB"."ABFV-207 FEED BACK OPEN" )
      Contact( "INPUT MAPPING DB"."ABFV 204 FEED BACK OPEN" )
      Contact( "INPUT MAPPING DB"."ABFV 203 FEED BACK OPEN" )
   END_RUNG wire#w1
   RUNG wire#powerrail
      { S7_Templates := "SrcType := Int" } EQ_Contact(in1 := "MODE SELECTION DB"."UF PLC_1 MODE BUFF", in2 := 1)
      { S7_Templates := "SrcType := Int" } EQ_Contact(in1 := "MODE SELECTION DB"."UF PLC_1 PROCESS BUFF", in2 := 880)
      Contact( "TIMING_SECS_DB_15".DONE )
      wire#w2
      Coil( "TIMING_SECS_DB_15".RESET )
   END_RUNG
   RUNG wire#w2
      Move(in := 885, out1 => "MODE SELECTION DB"."UF PLC_1 PROCESS BUFF")
   END_RUNG
   RUNG wire#powerrail
      { S7_Templates := "SrcType := Int" } EQ_Contact(in1 := "MODE SELECTION DB"."UF PLC_1 MODE BUFF", in2 := 1)
      { S7_Templates := "SrcType := Int" } EQ_Contact(in1 := "MODE SELECTION DB"."UF PLC_1 PROCESS BUFF", in2 := 885)
      { S7_Templates := "time_type := Time" } "IEC_Timer_0_DB_87".TON(pt := T#5s, et =>)
      Move(in := 890, out1 => "MODE SELECTION DB"."UF PLC_1 PROCESS BUFF")
   END_RUNG
   // the same network as SCL:
   "TIMING_SECS_DB_15"("SET TIME" := "CEB_2 DB".BACKWASH_1,   // "TIMING_SECS"
                       INPUT := ("MODE SELECTION DB"."UF PLC_1 MODE BUFF" = 1) AND ("MODE SELECTION DB"."UF PLC_1 PROCESS BUFF" = 880) AND "INPUT MAPPING DB"."ABFV-208 FEED BACK OPEN" AND "INPUT MAPPING DB"."ABFV-207 FEED BACK OPEN" AND "INPUT MAPPING DB"."ABFV 204 FEED BACK OPEN" AND "INPUT MAPPING DB"."ABFV 203 FEED BACK OPEN",
                       "PRESENT VALUE OF TIME" => "CEB_2 DB".PV.BACKWASH_1);
   "TIMING_SECS_DB_15".RESET := ("MODE SELECTION DB"."UF PLC_1 MODE BUFF" = 1) AND ("MODE SELECTION DB"."UF PLC_1 PROCESS BUFF" = 880) AND "TIMING_SECS_DB_15".DONE;
   IF "TIMING_SECS_DB_15".RESET THEN "MODE SELECTION DB"."UF PLC_1 PROCESS BUFF" := 885; END_IF;
   "IEC_Timer_0_DB_87".TON(IN := ("MODE SELECTION DB"."UF PLC_1 MODE BUFF" = 1) AND ("MODE SELECTION DB"."UF PLC_1 PROCESS BUFF" = 885),
                           PT := T#5s);
   IF "IEC_Timer_0_DB_87".Q THEN "MODE SELECTION DB"."UF PLC_1 PROCESS BUFF" := 890; END_IF;
END_REGION

REGION Network 41: ABFV 208 CLOSE FB
   RUNG wire#powerrail
      { S7_Templates := "SrcType := Int" } EQ_Contact(in1 := "MODE SELECTION DB"."UF PLC_1 MODE BUFF", in2 := 1)
      { S7_Templates := "SrcType := Int" } EQ_Contact(in1 := "MODE SELECTION DB"."UF PLC_1 PROCESS BUFF", in2 := 890)
      Move(in := 895, out1 => "MODE SELECTION DB"."UF PLC_1 PROCESS BUFF")
   END_RUNG
   // the same network as SCL:
   IF ("MODE SELECTION DB"."UF PLC_1 MODE BUFF" = 1) AND ("MODE SELECTION DB"."UF PLC_1 PROCESS BUFF" = 890) THEN
       "MODE SELECTION DB"."UF PLC_1 PROCESS BUFF" := 895;
   END_IF;
END_REGION

REGION Network 42: ABFV 207 CLOSE FB
   RUNG wire#powerrail
      { S7_Templates := "SrcType := Int" } EQ_Contact(in1 := "MODE SELECTION DB"."UF PLC_1 MODE BUFF", in2 := 1)
      { S7_Templates := "SrcType := Int" } EQ_Contact(in1 := "MODE SELECTION DB"."UF PLC_1 PROCESS BUFF", in2 := 895)
      Move(in := 900, out1 => "MODE SELECTION DB"."UF PLC_1 PROCESS BUFF")
   END_RUNG
   // the same network as SCL:
   IF ("MODE SELECTION DB"."UF PLC_1 MODE BUFF" = 1) AND ("MODE SELECTION DB"."UF PLC_1 PROCESS BUFF" = 895) THEN
       "MODE SELECTION DB"."UF PLC_1 PROCESS BUFF" := 900;
   END_IF;
END_REGION

REGION Network 43: ABFV 204 CLOSE FB
   RUNG wire#powerrail
      { S7_Templates := "SrcType := Int" } EQ_Contact(in1 := "MODE SELECTION DB"."UF PLC_1 MODE BUFF", in2 := 1)
      { S7_Templates := "SrcType := Int" } EQ_Contact(in1 := "MODE SELECTION DB"."UF PLC_1 PROCESS BUFF", in2 := 900)
      Move(in := 905, out1 => "MODE SELECTION DB"."UF PLC_1 PROCESS BUFF")
   END_RUNG
   // the same network as SCL:
   IF ("MODE SELECTION DB"."UF PLC_1 MODE BUFF" = 1) AND ("MODE SELECTION DB"."UF PLC_1 PROCESS BUFF" = 900) THEN
       "MODE SELECTION DB"."UF PLC_1 PROCESS BUFF" := 905;
   END_IF;
END_REGION

REGION Network 44: ABFV 203 CLOSE FB
   RUNG wire#powerrail
      { S7_Templates := "SrcType := Int" } EQ_Contact(in1 := "MODE SELECTION DB"."UF PLC_1 MODE BUFF", in2 := 1)
      { S7_Templates := "SrcType := Int" } EQ_Contact(in1 := "MODE SELECTION DB"."UF PLC_1 PROCESS BUFF", in2 := 905)
      Move(in := 910, out1 => "MODE SELECTION DB"."UF PLC_1 PROCESS BUFF")
   END_RUNG
   // the same network as SCL:
   IF ("MODE SELECTION DB"."UF PLC_1 MODE BUFF" = 1) AND ("MODE SELECTION DB"."UF PLC_1 PROCESS BUFF" = 905) THEN
       "MODE SELECTION DB"."UF PLC_1 PROCESS BUFF" := 910;
   END_IF;
END_REGION

REGION Network 45: 915
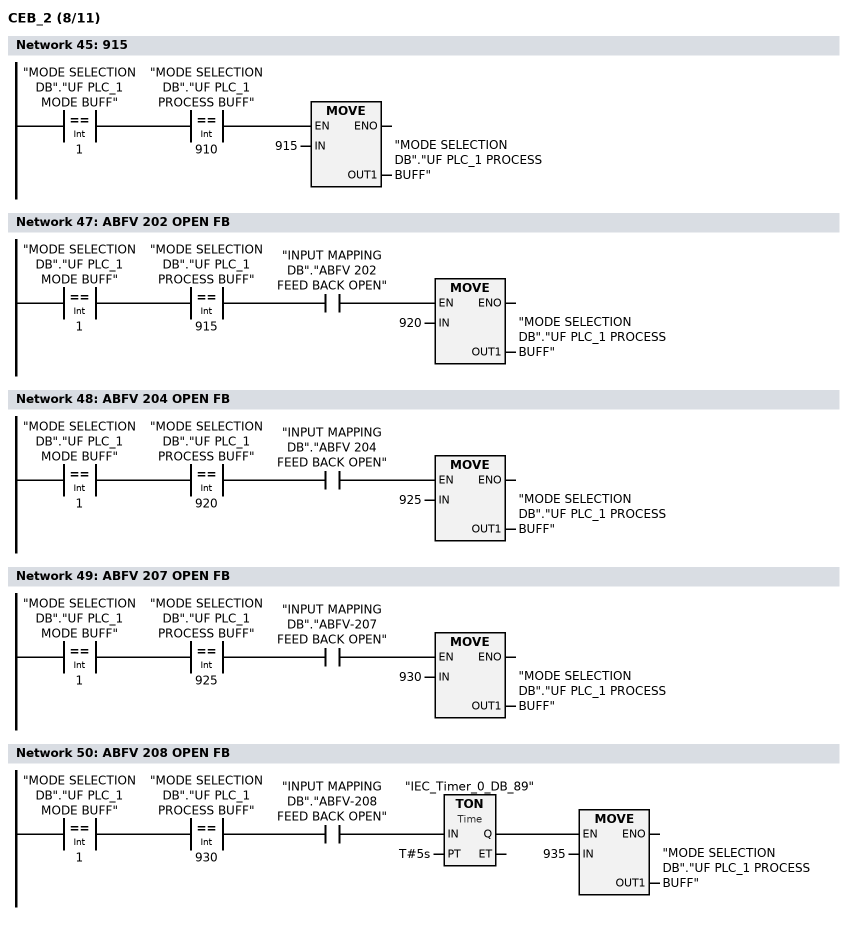
   RUNG wire#powerrail
      { S7_Templates := "SrcType := Int" } EQ_Contact(in1 := "MODE SELECTION DB"."UF PLC_1 MODE BUFF", in2 := 1)
      { S7_Templates := "SrcType := Int" } EQ_Contact(in1 := "MODE SELECTION DB"."UF PLC_1 PROCESS BUFF", in2 := 910)
      Move(in := 915, out1 => "MODE SELECTION DB"."UF PLC_1 PROCESS BUFF")
   END_RUNG
   // the same network as SCL:
   IF ("MODE SELECTION DB"."UF PLC_1 MODE BUFF" = 1) AND ("MODE SELECTION DB"."UF PLC_1 PROCESS BUFF" = 910) THEN
       "MODE SELECTION DB"."UF PLC_1 PROCESS BUFF" := 915;
   END_IF;
END_REGION

REGION Network 47: ABFV 202 OPEN FB
   RUNG wire#powerrail
      { S7_Templates := "SrcType := Int" } EQ_Contact(in1 := "MODE SELECTION DB"."UF PLC_1 MODE BUFF", in2 := 1)
      { S7_Templates := "SrcType := Int" } EQ_Contact(in1 := "MODE SELECTION DB"."UF PLC_1 PROCESS BUFF", in2 := 915)
      Contact( "INPUT MAPPING DB"."ABFV 202 FEED BACK OPEN" )
      Move(in := 920, out1 => "MODE SELECTION DB"."UF PLC_1 PROCESS BUFF")
   END_RUNG
   // the same network as SCL:
   IF ("MODE SELECTION DB"."UF PLC_1 MODE BUFF" = 1) AND ("MODE SELECTION DB"."UF PLC_1 PROCESS BUFF" = 915) AND "INPUT MAPPING DB"."ABFV 202 FEED BACK OPEN" THEN
       "MODE SELECTION DB"."UF PLC_1 PROCESS BUFF" := 920;
   END_IF;
END_REGION

REGION Network 48: ABFV 204 OPEN FB
   RUNG wire#powerrail
      { S7_Templates := "SrcType := Int" } EQ_Contact(in1 := "MODE SELECTION DB"."UF PLC_1 MODE BUFF", in2 := 1)
      { S7_Templates := "SrcType := Int" } EQ_Contact(in1 := "MODE SELECTION DB"."UF PLC_1 PROCESS BUFF", in2 := 920)
      Contact( "INPUT MAPPING DB"."ABFV 204 FEED BACK OPEN" )
      Move(in := 925, out1 => "MODE SELECTION DB"."UF PLC_1 PROCESS BUFF")
   END_RUNG
   // the same network as SCL:
   IF ("MODE SELECTION DB"."UF PLC_1 MODE BUFF" = 1) AND ("MODE SELECTION DB"."UF PLC_1 PROCESS BUFF" = 920) AND "INPUT MAPPING DB"."ABFV 204 FEED BACK OPEN" THEN
       "MODE SELECTION DB"."UF PLC_1 PROCESS BUFF" := 925;
   END_IF;
END_REGION

REGION Network 49: ABFV 207 OPEN FB
   RUNG wire#powerrail
      { S7_Templates := "SrcType := Int" } EQ_Contact(in1 := "MODE SELECTION DB"."UF PLC_1 MODE BUFF", in2 := 1)
      { S7_Templates := "SrcType := Int" } EQ_Contact(in1 := "MODE SELECTION DB"."UF PLC_1 PROCESS BUFF", in2 := 925)
      Contact( "INPUT MAPPING DB"."ABFV-207 FEED BACK OPEN" )
      Move(in := 930, out1 => "MODE SELECTION DB"."UF PLC_1 PROCESS BUFF")
   END_RUNG
   // the same network as SCL:
   IF ("MODE SELECTION DB"."UF PLC_1 MODE BUFF" = 1) AND ("MODE SELECTION DB"."UF PLC_1 PROCESS BUFF" = 925) AND "INPUT MAPPING DB"."ABFV-207 FEED BACK OPEN" THEN
       "MODE SELECTION DB"."UF PLC_1 PROCESS BUFF" := 930;
   END_IF;
END_REGION

REGION Network 50: ABFV 208 OPEN FB
   RUNG wire#powerrail
      { S7_Templates := "SrcType := Int" } EQ_Contact(in1 := "MODE SELECTION DB"."UF PLC_1 MODE BUFF", in2 := 1)
      { S7_Templates := "SrcType := Int" } EQ_Contact(in1 := "MODE SELECTION DB"."UF PLC_1 PROCESS BUFF", in2 := 930)
      Contact( "INPUT MAPPING DB"."ABFV-208 FEED BACK OPEN" )
      { S7_Templates := "time_type := Time" } "IEC_Timer_0_DB_89".TON(pt := T#5s, et =>)
      Move(in := 935, out1 => "MODE SELECTION DB"."UF PLC_1 PROCESS BUFF")
   END_RUNG
   // the same network as SCL:
   "IEC_Timer_0_DB_89".TON(IN := ("MODE SELECTION DB"."UF PLC_1 MODE BUFF" = 1) AND ("MODE SELECTION DB"."UF PLC_1 PROCESS BUFF" = 930) AND "INPUT MAPPING DB"."ABFV-208 FEED BACK OPEN",
                           PT := T#5s);
   IF "IEC_Timer_0_DB_89".Q THEN "MODE SELECTION DB"."UF PLC_1 PROCESS BUFF" := 935; END_IF;
END_REGION

REGION Network 51: BACKWASH_2
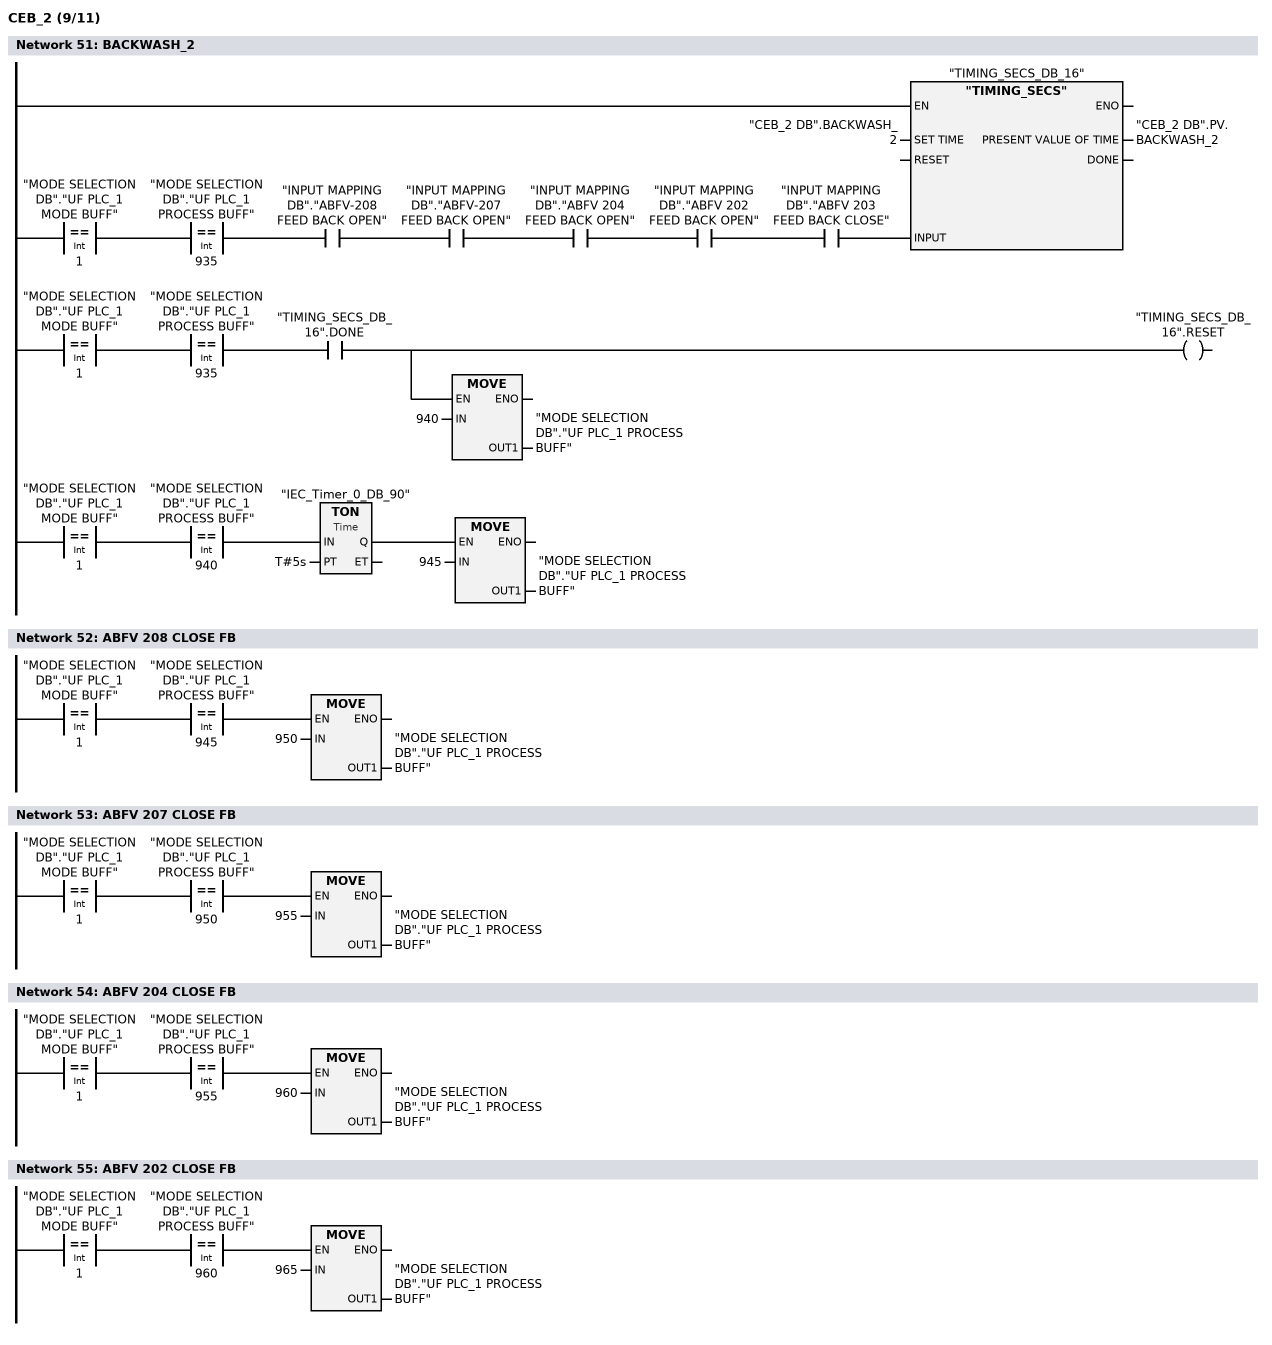
   RUNG wire#powerrail
      "TIMING_SECS_DB_16"(INPUT := wire#w1, "SET TIME" := "CEB_2 DB".BACKWASH_2, RESET :=, "PRESENT VALUE OF TIME" => "CEB_2 DB".PV.BACKWASH_2, DONE =>)
   END_RUNG
   RUNG wire#powerrail
      { S7_Templates := "SrcType := Int" } EQ_Contact(in1 := "MODE SELECTION DB"."UF PLC_1 MODE BUFF", in2 := 1)
      { S7_Templates := "SrcType := Int" } EQ_Contact(in1 := "MODE SELECTION DB"."UF PLC_1 PROCESS BUFF", in2 := 935)
      Contact( "INPUT MAPPING DB"."ABFV-208 FEED BACK OPEN" )
      Contact( "INPUT MAPPING DB"."ABFV-207 FEED BACK OPEN" )
      Contact( "INPUT MAPPING DB"."ABFV 204 FEED BACK OPEN" )
      Contact( "INPUT MAPPING DB"."ABFV 202 FEED BACK OPEN" )
      Contact( "INPUT MAPPING DB"."ABFV 203 FEED BACK CLOSE" )
   END_RUNG wire#w1
   RUNG wire#powerrail
      { S7_Templates := "SrcType := Int" } EQ_Contact(in1 := "MODE SELECTION DB"."UF PLC_1 MODE BUFF", in2 := 1)
      { S7_Templates := "SrcType := Int" } EQ_Contact(in1 := "MODE SELECTION DB"."UF PLC_1 PROCESS BUFF", in2 := 935)
      Contact( "TIMING_SECS_DB_16".DONE )
      wire#w2
      Coil( "TIMING_SECS_DB_16".RESET )
   END_RUNG
   RUNG wire#w2
      Move(in := 940, out1 => "MODE SELECTION DB"."UF PLC_1 PROCESS BUFF")
   END_RUNG
   RUNG wire#powerrail
      { S7_Templates := "SrcType := Int" } EQ_Contact(in1 := "MODE SELECTION DB"."UF PLC_1 MODE BUFF", in2 := 1)
      { S7_Templates := "SrcType := Int" } EQ_Contact(in1 := "MODE SELECTION DB"."UF PLC_1 PROCESS BUFF", in2 := 940)
      { S7_Templates := "time_type := Time" } "IEC_Timer_0_DB_90".TON(pt := T#5s, et =>)
      Move(in := 945, out1 => "MODE SELECTION DB"."UF PLC_1 PROCESS BUFF")
   END_RUNG
   // the same network as SCL:
   "TIMING_SECS_DB_16"("SET TIME" := "CEB_2 DB".BACKWASH_2,   // "TIMING_SECS"
                       INPUT := ("MODE SELECTION DB"."UF PLC_1 MODE BUFF" = 1) AND ("MODE SELECTION DB"."UF PLC_1 PROCESS BUFF" = 935) AND "INPUT MAPPING DB"."ABFV-208 FEED BACK OPEN" AND "INPUT MAPPING DB"."ABFV-207 FEED BACK OPEN" AND "INPUT MAPPING DB"."ABFV 204 FEED BACK OPEN" AND "INPUT MAPPING DB"."ABFV 202 FEED BACK OPEN" AND "INPUT MAPPING DB"."ABFV 203 FEED BACK CLOSE",
                       "PRESENT VALUE OF TIME" => "CEB_2 DB".PV.BACKWASH_2);
   "TIMING_SECS_DB_16".RESET := ("MODE SELECTION DB"."UF PLC_1 MODE BUFF" = 1) AND ("MODE SELECTION DB"."UF PLC_1 PROCESS BUFF" = 935) AND "TIMING_SECS_DB_16".DONE;
   IF "TIMING_SECS_DB_16".RESET THEN "MODE SELECTION DB"."UF PLC_1 PROCESS BUFF" := 940; END_IF;
   "IEC_Timer_0_DB_90".TON(IN := ("MODE SELECTION DB"."UF PLC_1 MODE BUFF" = 1) AND ("MODE SELECTION DB"."UF PLC_1 PROCESS BUFF" = 940),
                           PT := T#5s);
   IF "IEC_Timer_0_DB_90".Q THEN "MODE SELECTION DB"."UF PLC_1 PROCESS BUFF" := 945; END_IF;
END_REGION

REGION Network 52: ABFV 208 CLOSE FB
   RUNG wire#powerrail
      { S7_Templates := "SrcType := Int" } EQ_Contact(in1 := "MODE SELECTION DB"."UF PLC_1 MODE BUFF", in2 := 1)
      { S7_Templates := "SrcType := Int" } EQ_Contact(in1 := "MODE SELECTION DB"."UF PLC_1 PROCESS BUFF", in2 := 945)
      Move(in := 950, out1 => "MODE SELECTION DB"."UF PLC_1 PROCESS BUFF")
   END_RUNG
   // the same network as SCL:
   IF ("MODE SELECTION DB"."UF PLC_1 MODE BUFF" = 1) AND ("MODE SELECTION DB"."UF PLC_1 PROCESS BUFF" = 945) THEN
       "MODE SELECTION DB"."UF PLC_1 PROCESS BUFF" := 950;
   END_IF;
END_REGION

REGION Network 53: ABFV 207 CLOSE FB
   RUNG wire#powerrail
      { S7_Templates := "SrcType := Int" } EQ_Contact(in1 := "MODE SELECTION DB"."UF PLC_1 MODE BUFF", in2 := 1)
      { S7_Templates := "SrcType := Int" } EQ_Contact(in1 := "MODE SELECTION DB"."UF PLC_1 PROCESS BUFF", in2 := 950)
      Move(in := 955, out1 => "MODE SELECTION DB"."UF PLC_1 PROCESS BUFF")
   END_RUNG
   // the same network as SCL:
   IF ("MODE SELECTION DB"."UF PLC_1 MODE BUFF" = 1) AND ("MODE SELECTION DB"."UF PLC_1 PROCESS BUFF" = 950) THEN
       "MODE SELECTION DB"."UF PLC_1 PROCESS BUFF" := 955;
   END_IF;
END_REGION

REGION Network 54: ABFV 204 CLOSE FB
   RUNG wire#powerrail
      { S7_Templates := "SrcType := Int" } EQ_Contact(in1 := "MODE SELECTION DB"."UF PLC_1 MODE BUFF", in2 := 1)
      { S7_Templates := "SrcType := Int" } EQ_Contact(in1 := "MODE SELECTION DB"."UF PLC_1 PROCESS BUFF", in2 := 955)
      Move(in := 960, out1 => "MODE SELECTION DB"."UF PLC_1 PROCESS BUFF")
   END_RUNG
   // the same network as SCL:
   IF ("MODE SELECTION DB"."UF PLC_1 MODE BUFF" = 1) AND ("MODE SELECTION DB"."UF PLC_1 PROCESS BUFF" = 955) THEN
       "MODE SELECTION DB"."UF PLC_1 PROCESS BUFF" := 960;
   END_IF;
END_REGION

REGION Network 55: ABFV 202 CLOSE FB
   RUNG wire#powerrail
      { S7_Templates := "SrcType := Int" } EQ_Contact(in1 := "MODE SELECTION DB"."UF PLC_1 MODE BUFF", in2 := 1)
      { S7_Templates := "SrcType := Int" } EQ_Contact(in1 := "MODE SELECTION DB"."UF PLC_1 PROCESS BUFF", in2 := 960)
      Move(in := 965, out1 => "MODE SELECTION DB"."UF PLC_1 PROCESS BUFF")
   END_RUNG
   // the same network as SCL:
   IF ("MODE SELECTION DB"."UF PLC_1 MODE BUFF" = 1) AND ("MODE SELECTION DB"."UF PLC_1 PROCESS BUFF" = 960) THEN
       "MODE SELECTION DB"."UF PLC_1 PROCESS BUFF" := 965;
   END_IF;
END_REGION

REGION Network 56: 970
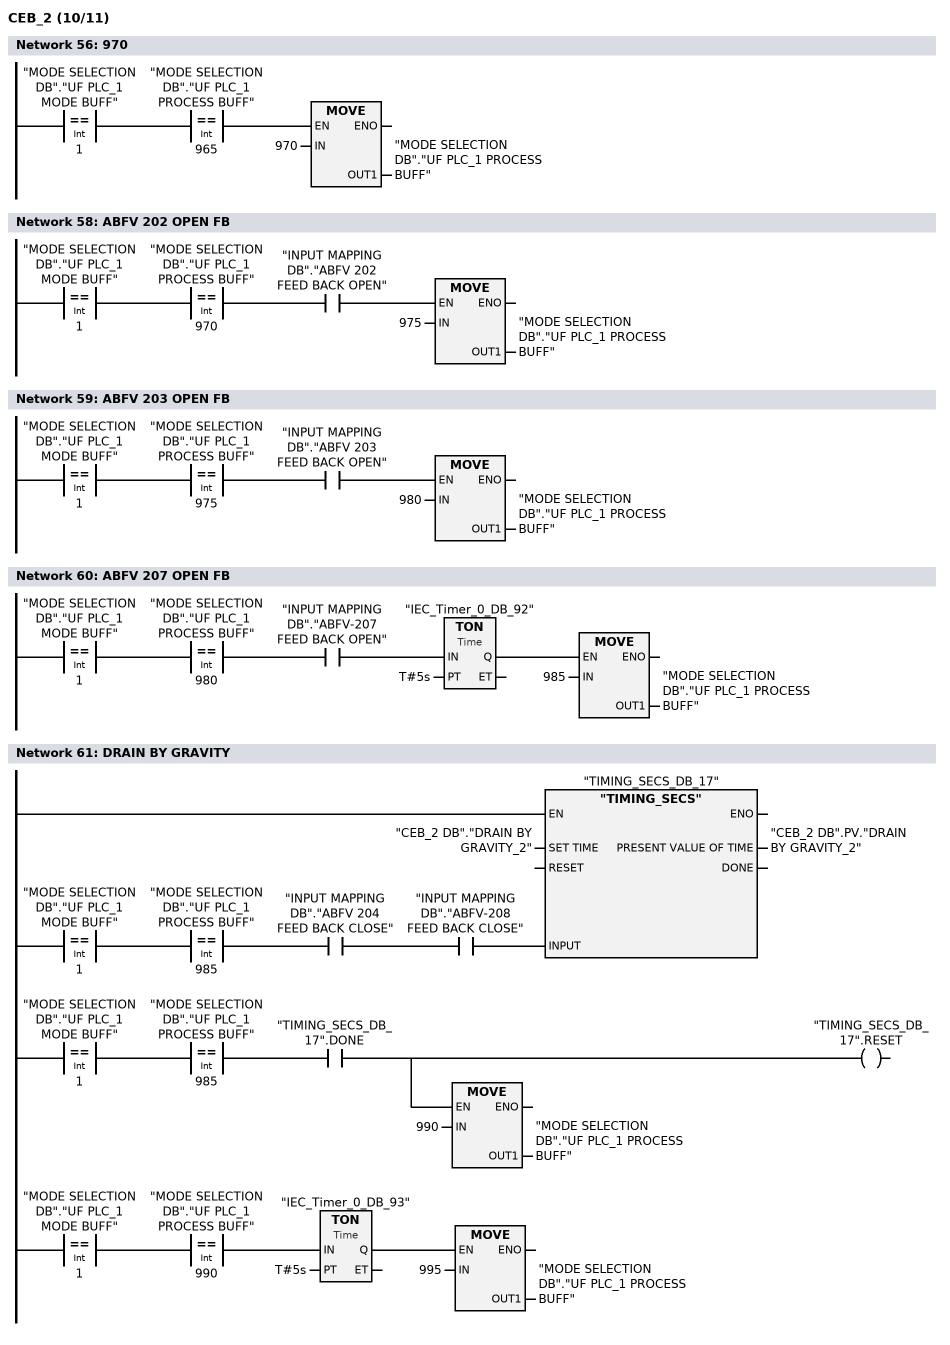
   RUNG wire#powerrail
      { S7_Templates := "SrcType := Int" } EQ_Contact(in1 := "MODE SELECTION DB"."UF PLC_1 MODE BUFF", in2 := 1)
      { S7_Templates := "SrcType := Int" } EQ_Contact(in1 := "MODE SELECTION DB"."UF PLC_1 PROCESS BUFF", in2 := 965)
      Move(in := 970, out1 => "MODE SELECTION DB"."UF PLC_1 PROCESS BUFF")
   END_RUNG
   // the same network as SCL:
   IF ("MODE SELECTION DB"."UF PLC_1 MODE BUFF" = 1) AND ("MODE SELECTION DB"."UF PLC_1 PROCESS BUFF" = 965) THEN
       "MODE SELECTION DB"."UF PLC_1 PROCESS BUFF" := 970;
   END_IF;
END_REGION

REGION Network 58: ABFV 202 OPEN FB
   RUNG wire#powerrail
      { S7_Templates := "SrcType := Int" } EQ_Contact(in1 := "MODE SELECTION DB"."UF PLC_1 MODE BUFF", in2 := 1)
      { S7_Templates := "SrcType := Int" } EQ_Contact(in1 := "MODE SELECTION DB"."UF PLC_1 PROCESS BUFF", in2 := 970)
      Contact( "INPUT MAPPING DB"."ABFV 202 FEED BACK OPEN" )
      Move(in := 975, out1 => "MODE SELECTION DB"."UF PLC_1 PROCESS BUFF")
   END_RUNG
   // the same network as SCL:
   IF ("MODE SELECTION DB"."UF PLC_1 MODE BUFF" = 1) AND ("MODE SELECTION DB"."UF PLC_1 PROCESS BUFF" = 970) AND "INPUT MAPPING DB"."ABFV 202 FEED BACK OPEN" THEN
       "MODE SELECTION DB"."UF PLC_1 PROCESS BUFF" := 975;
   END_IF;
END_REGION

REGION Network 59: ABFV 203 OPEN FB
   RUNG wire#powerrail
      { S7_Templates := "SrcType := Int" } EQ_Contact(in1 := "MODE SELECTION DB"."UF PLC_1 MODE BUFF", in2 := 1)
      { S7_Templates := "SrcType := Int" } EQ_Contact(in1 := "MODE SELECTION DB"."UF PLC_1 PROCESS BUFF", in2 := 975)
      Contact( "INPUT MAPPING DB"."ABFV 203 FEED BACK OPEN" )
      Move(in := 980, out1 => "MODE SELECTION DB"."UF PLC_1 PROCESS BUFF")
   END_RUNG
   // the same network as SCL:
   IF ("MODE SELECTION DB"."UF PLC_1 MODE BUFF" = 1) AND ("MODE SELECTION DB"."UF PLC_1 PROCESS BUFF" = 975) AND "INPUT MAPPING DB"."ABFV 203 FEED BACK OPEN" THEN
       "MODE SELECTION DB"."UF PLC_1 PROCESS BUFF" := 980;
   END_IF;
END_REGION

REGION Network 60: ABFV 207 OPEN FB
   RUNG wire#powerrail
      { S7_Templates := "SrcType := Int" } EQ_Contact(in1 := "MODE SELECTION DB"."UF PLC_1 MODE BUFF", in2 := 1)
      { S7_Templates := "SrcType := Int" } EQ_Contact(in1 := "MODE SELECTION DB"."UF PLC_1 PROCESS BUFF", in2 := 980)
      Contact( "INPUT MAPPING DB"."ABFV-207 FEED BACK OPEN" )
      { S7_Templates := "time_type := Time" } "IEC_Timer_0_DB_92".TON(pt := T#5s, et =>)
      Move(in := 985, out1 => "MODE SELECTION DB"."UF PLC_1 PROCESS BUFF")
   END_RUNG
   // the same network as SCL:
   "IEC_Timer_0_DB_92".TON(IN := ("MODE SELECTION DB"."UF PLC_1 MODE BUFF" = 1) AND ("MODE SELECTION DB"."UF PLC_1 PROCESS BUFF" = 980) AND "INPUT MAPPING DB"."ABFV-207 FEED BACK OPEN",
                           PT := T#5s);
   IF "IEC_Timer_0_DB_92".Q THEN "MODE SELECTION DB"."UF PLC_1 PROCESS BUFF" := 985; END_IF;
END_REGION

REGION Network 61: DRAIN BY GRAVITY
   RUNG wire#powerrail
      "TIMING_SECS_DB_17"(INPUT := wire#w1, "SET TIME" := "CEB_2 DB"."DRAIN BY GRAVITY_2", RESET :=, "PRESENT VALUE OF TIME" => "CEB_2 DB".PV."DRAIN BY GRAVITY_2", DONE =>)
   END_RUNG
   RUNG wire#powerrail
      { S7_Templates := "SrcType := Int" } EQ_Contact(in1 := "MODE SELECTION DB"."UF PLC_1 MODE BUFF", in2 := 1)
      { S7_Templates := "SrcType := Int" } EQ_Contact(in1 := "MODE SELECTION DB"."UF PLC_1 PROCESS BUFF", in2 := 985)
      Contact( "INPUT MAPPING DB"."ABFV 204 FEED BACK CLOSE" )
      Contact( "INPUT MAPPING DB"."ABFV-208 FEED BACK CLOSE" )
   END_RUNG wire#w1
   RUNG wire#powerrail
      { S7_Templates := "SrcType := Int" } EQ_Contact(in1 := "MODE SELECTION DB"."UF PLC_1 MODE BUFF", in2 := 1)
      { S7_Templates := "SrcType := Int" } EQ_Contact(in1 := "MODE SELECTION DB"."UF PLC_1 PROCESS BUFF", in2 := 985)
      Contact( "TIMING_SECS_DB_17".DONE )
      wire#w2
      Coil( "TIMING_SECS_DB_17".RESET )
   END_RUNG
   RUNG wire#w2
      Move(in := 990, out1 => "MODE SELECTION DB"."UF PLC_1 PROCESS BUFF")
   END_RUNG
   RUNG wire#powerrail
      { S7_Templates := "SrcType := Int" } EQ_Contact(in1 := "MODE SELECTION DB"."UF PLC_1 MODE BUFF", in2 := 1)
      { S7_Templates := "SrcType := Int" } EQ_Contact(in1 := "MODE SELECTION DB"."UF PLC_1 PROCESS BUFF", in2 := 990)
      { S7_Templates := "time_type := Time" } "IEC_Timer_0_DB_93".TON(pt := T#5s, et =>)
      Move(in := 995, out1 => "MODE SELECTION DB"."UF PLC_1 PROCESS BUFF")
   END_RUNG
   // the same network as SCL:
   "TIMING_SECS_DB_17"("SET TIME" := "CEB_2 DB"."DRAIN BY GRAVITY_2",   // "TIMING_SECS"
                       INPUT := ("MODE SELECTION DB"."UF PLC_1 MODE BUFF" = 1) AND ("MODE SELECTION DB"."UF PLC_1 PROCESS BUFF" = 985) AND "INPUT MAPPING DB"."ABFV 204 FEED BACK CLOSE" AND "INPUT MAPPING DB"."ABFV-208 FEED BACK CLOSE",
                       "PRESENT VALUE OF TIME" => "CEB_2 DB".PV."DRAIN BY GRAVITY_2");
   "TIMING_SECS_DB_17".RESET := ("MODE SELECTION DB"."UF PLC_1 MODE BUFF" = 1) AND ("MODE SELECTION DB"."UF PLC_1 PROCESS BUFF" = 985) AND "TIMING_SECS_DB_17".DONE;
   IF "TIMING_SECS_DB_17".RESET THEN "MODE SELECTION DB"."UF PLC_1 PROCESS BUFF" := 990; END_IF;
   "IEC_Timer_0_DB_93".TON(IN := ("MODE SELECTION DB"."UF PLC_1 MODE BUFF" = 1) AND ("MODE SELECTION DB"."UF PLC_1 PROCESS BUFF" = 990),
                           PT := T#5s);
   IF "IEC_Timer_0_DB_93".Q THEN "MODE SELECTION DB"."UF PLC_1 PROCESS BUFF" := 995; END_IF;
END_REGION

REGION Network 62: ABFV 207 CLOSE FB
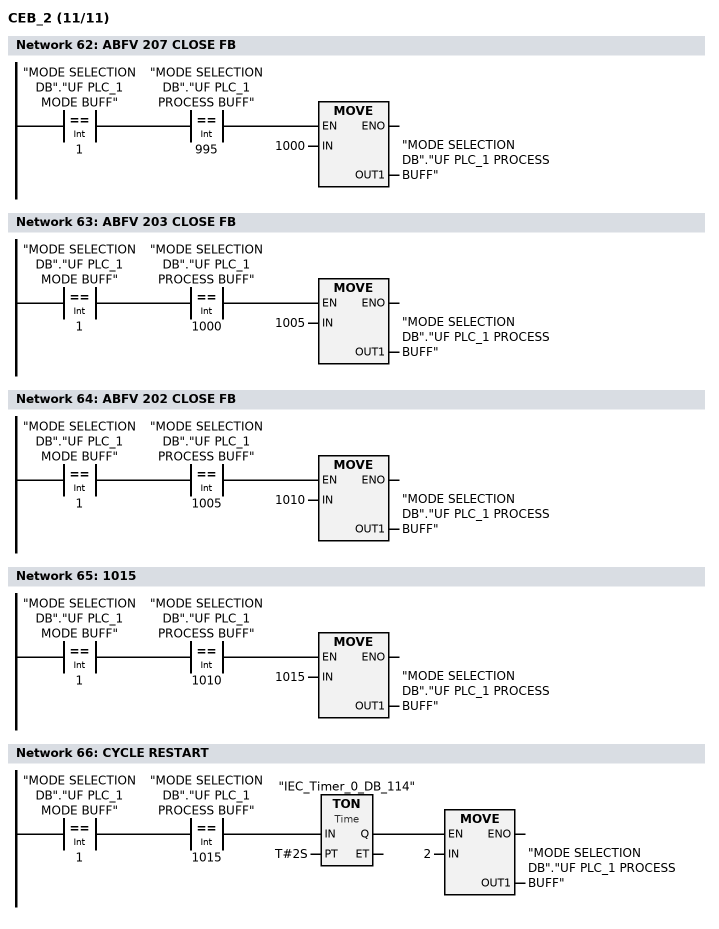
   RUNG wire#powerrail
      { S7_Templates := "SrcType := Int" } EQ_Contact(in1 := "MODE SELECTION DB"."UF PLC_1 MODE BUFF", in2 := 1)
      { S7_Templates := "SrcType := Int" } EQ_Contact(in1 := "MODE SELECTION DB"."UF PLC_1 PROCESS BUFF", in2 := 995)
      Move(in := 1000, out1 => "MODE SELECTION DB"."UF PLC_1 PROCESS BUFF")
   END_RUNG
   // the same network as SCL:
   IF ("MODE SELECTION DB"."UF PLC_1 MODE BUFF" = 1) AND ("MODE SELECTION DB"."UF PLC_1 PROCESS BUFF" = 995) THEN
       "MODE SELECTION DB"."UF PLC_1 PROCESS BUFF" := 1000;
   END_IF;
END_REGION

REGION Network 63: ABFV 203 CLOSE FB
   RUNG wire#powerrail
      { S7_Templates := "SrcType := Int" } EQ_Contact(in1 := "MODE SELECTION DB"."UF PLC_1 MODE BUFF", in2 := 1)
      { S7_Templates := "SrcType := Int" } EQ_Contact(in1 := "MODE SELECTION DB"."UF PLC_1 PROCESS BUFF", in2 := 1000)
      Move(in := 1005, out1 => "MODE SELECTION DB"."UF PLC_1 PROCESS BUFF")
   END_RUNG
   // the same network as SCL:
   IF ("MODE SELECTION DB"."UF PLC_1 MODE BUFF" = 1) AND ("MODE SELECTION DB"."UF PLC_1 PROCESS BUFF" = 1000) THEN
       "MODE SELECTION DB"."UF PLC_1 PROCESS BUFF" := 1005;
   END_IF;
END_REGION

REGION Network 64: ABFV 202 CLOSE FB
   RUNG wire#powerrail
      { S7_Templates := "SrcType := Int" } EQ_Contact(in1 := "MODE SELECTION DB"."UF PLC_1 MODE BUFF", in2 := 1)
      { S7_Templates := "SrcType := Int" } EQ_Contact(in1 := "MODE SELECTION DB"."UF PLC_1 PROCESS BUFF", in2 := 1005)
      Move(in := 1010, out1 => "MODE SELECTION DB"."UF PLC_1 PROCESS BUFF")
   END_RUNG
   // the same network as SCL:
   IF ("MODE SELECTION DB"."UF PLC_1 MODE BUFF" = 1) AND ("MODE SELECTION DB"."UF PLC_1 PROCESS BUFF" = 1005) THEN
       "MODE SELECTION DB"."UF PLC_1 PROCESS BUFF" := 1010;
   END_IF;
END_REGION

REGION Network 65: 1015
   RUNG wire#powerrail
      { S7_Templates := "SrcType := Int" } EQ_Contact(in1 := "MODE SELECTION DB"."UF PLC_1 MODE BUFF", in2 := 1)
      { S7_Templates := "SrcType := Int" } EQ_Contact(in1 := "MODE SELECTION DB"."UF PLC_1 PROCESS BUFF", in2 := 1010)
      Move(in := 1015, out1 => "MODE SELECTION DB"."UF PLC_1 PROCESS BUFF")
   END_RUNG
   // the same network as SCL:
   IF ("MODE SELECTION DB"."UF PLC_1 MODE BUFF" = 1) AND ("MODE SELECTION DB"."UF PLC_1 PROCESS BUFF" = 1010) THEN
       "MODE SELECTION DB"."UF PLC_1 PROCESS BUFF" := 1015;
   END_IF;
END_REGION

REGION Network 66: CYCLE RESTART
   RUNG wire#powerrail
      { S7_Templates := "SrcType := Int" } EQ_Contact(in1 := "MODE SELECTION DB"."UF PLC_1 MODE BUFF", in2 := 1)
      { S7_Templates := "SrcType := Int" } EQ_Contact(in1 := "MODE SELECTION DB"."UF PLC_1 PROCESS BUFF", in2 := 1015)
      { S7_Templates := "time_type := Time" } "IEC_Timer_0_DB_114".TON(pt := T#2S, et =>)
      Move(in := 2, out1 => "MODE SELECTION DB"."UF PLC_1 PROCESS BUFF")
   END_RUNG
   // the same network as SCL:
   "IEC_Timer_0_DB_114".TON(IN := ("MODE SELECTION DB"."UF PLC_1 MODE BUFF" = 1) AND ("MODE SELECTION DB"."UF PLC_1 PROCESS BUFF" = 1015),
                           PT := T#2S);
   IF "IEC_Timer_0_DB_114".Q THEN "MODE SELECTION DB"."UF PLC_1 PROCESS BUFF" := 2; END_IF;
END_REGION
END_FUNCTION
